	REGION Główny błąd - wszystkie pętle nie działają
	  //kasowanie wartości zmiennych errorStatus odblokowanie magistrali
	  IF "setErrorModbsmasterABB_1" AND "setErrorModbsmasterFal" THEN
	    //ustaw znacznik błędu
	    "db10datablock".setRTU_Error := TRUE;
	    // resetuj mdbusMastererror dla wszystkich pętli
	    "dbTags_master_Fal_1".modbusMaster.error := FALSE;
	    "dbTags_master_ABB_1".modbusMaster.error := FALSE;
	    
	  ELSE
	    "db10datablock".setRTU_Error := FALSE;
	    ;
	  END_IF;
	  
	END_REGION
	
	IF ("db10datablock".RTU_Fal_1errorStatus = 0) AND ("db10datablock".RTU_MPP04_1errorStatus = 0) THEN
	  // kasowanie znacznika błędu komunikacj modbus rtu
	  "db10datablock".setRTU_Error := FALSE;
	  ;
	END_IF;
	
	
	
	
	
	REGION Falownik Modbau RTU
	  // Sprawdzanie czy 
	  IF "dbTags_master_Fal_1".step = 27 THEN
	    // Statement section IF
	    "dbTags_master_Fal_1".modbusMaster.error := FALSE;
	    "dbTags_master_Fal_1".modbusMaster.busy := FALSE;
	    "dbTags_master_Fal_1".modbusMaster.status:= 0;
	    
	   
	   // jeśli MPP04_1 kod błedu 80C8 (brak urządzenia na linni) to uruchom pętlę modbus dla falownika
	    IF "dbTags_master_ABB_1".modbusMaster.status = 16#80C8 AND ("dbTags_master_Fal_1".step = 27 OR "dbTags_master_Fal_1".step = 25 )
	    THEN
	      // Statement section 
	      "setErrorModbsmasterFal" := FALSE;
	      "dbTags_master_Fal_1".step := 1;
	      
	      ;
	    END_IF;
	    
	    ;
	  END_IF;
	  
	  // awaria komunikacji z falownikiem Modbus-RTU
	  IF "setErrorModbsmasterFal" THEN
	    // ustaw bit awarii 
	    "dbmanagement".sterowanie_1.awaria_modbus_falownik:= TRUE
	    ;
	  END_IF;
	  
	  // kasowanie biti awarii komunikacji falownika Modbus-RTU
	  IF "memStep_errorFal" = 100 THEN
	    // kasowanie
	    "dbmanagement".sterowanie_1.awaria_modbus_falownik:= FALSE
	    ;
	  END_IF;
	  
	  
	END_REGION
	
	REGION MPP04-1 Modbau RTU
	  // Sprawdzanie czy 
	  IF "dbTags_master_ABB_1".step = 27 AND "dbTags_master_Fal_1".step = 27
	     THEN
	    // 
	    "dbTags_master_ABB_1".modbusMaster.error := FALSE;
	    "dbTags_master_ABB_1".modbusMaster.busy := FALSE;
	    "dbTags_master_ABB_1".modbusMaster.status := 0;
	    "dbTags_master_Fal_1".step := 1;
	    
	    ;
	  END_IF;
	  
	  IF "dbTags_master_ABB_1".step = 27
	  THEN
	    // 
	    "dbTags_master_ABB_1".modbusMaster.error := FALSE;
	    "dbTags_master_ABB_1".modbusMaster.busy := FALSE;
	    "dbTags_master_ABB_1".modbusMaster.status := 0;
	    //"dbTags_master_MPP04_1".step := 25;
	    
	    ;
	  END_IF;
	  
	  
	  // awaria komunikacji z MPO04 Modbus-RTU
	  IF "setErrorModbsmasterABB_1"  THEN
	    // ustaw bit awarii po czasie zwłoki 
	    "IEC_Timer_errorRTU_histereza_DB".TON(IN:="setErrorModbsmasterABB_1",
	                                          PT:=T#30S);
	    #set_error_RTU := "IEC_Timer_errorRTU_histereza_DB".Q;
	    "dbmanagement".sterowanie_1.awaria_modbus_przepływ_pomp := #set_error_RTU;
	  ELSE
	    #set_error_RTU := FALSE;
	    ;
	  END_IF;
	  
	  // kasowanie biti awarii komunikacjiModbus-RTU
	  IF "memStep_errorMPP04-1" = 100  AND "setErrorModbsmasterABB_1" = FALSE THEN
	    // kasowanie
	    "dbmanagement".sterowanie_1.awaria_modbus_przepływ_pomp:= FALSE
	    ;
	  END_IF;
	  
	END_REGION
	
	
	
	//Modbus RTU Error Code RESET
	REGION Modbus RTU Error Code
	  // Ustaw reset modbus rtu
	  IF "db10datablock".RTU_stepRESET THEN
	    // Ustawienie domyślnych satrtowych 
	    "dbTags_master_ABB_1".step := 1;
	    
	    "dbTags_master_Fal_1".step := 25;
	    "dbTags_slave_RTU".step := 25;
	    
	    // Zerowanie kodu błędu
	    "dbTags_master_ABB_1".modbusMaster.errorStatus := 0;
	    "dbTags_master_Fal_1".modbusMaster.errorStatus := 0;
	    "dbTags_slave_RTU".modbusMaster.errorStatus := 0;
	    
	    "db10datablock".RTU_stepRESET := 0;
	    ;
	  END_IF;
	  
	  
	END_REGION
	
	// Ustawienie Błędu Modbus RTU 
	REGION Set Fault Modbus RTU 
	  // Jeśli zmienna kodu błędu różna od 0 to ustaw znacznik błędu Modbus w bloku danych SCADA
	  // i przekaż wartość błędów
	  IF "dbmanagement".sterowanie_1."alarm-modbus" = TRUE
	    
	  THEN
	    
	    "db10datablock".RTU_MPP04_1errorStatus := "dbTags_master_ABB_1".modbusMaster.errorStatus;
	    // Trzeba dopisać przekazanie błędu z PLC Zasuwy
	   // "DB10_instance_SCADA".RTU_MPP04_2errorStatus := "dbTags_master_MPP04_2".modbusMaster.errorStatus;
	    "db10datablock".RTU_Fal_1errorStatus := "dbTags_master_Fal_1".modbusMaster.errorStatus;
	    "db10datablock".RTU_MT101 := "dbTags_slave_RTU".modbusMaster.errorStatus;
	  ELSE
	    //
	    ;
	    ;
	  END_IF;
	  
	  
	  // Modbus przekaż bit do instancji SCADA Alarm ostrzeżenie kłoport z Modbau
	  // Przynajmniej jeden slave nie odpowiada
	  IF "dbTags_master_Fal_1".step = 27 OR "dbTags_master_ABB_1".step = 27 
	 
	  THEN
	    "dbmanagement".sterowanie_1."alarm-warning" := TRUE;
	
	    ;
	    
	  END_IF;
	  
	  IF "db10datablock".RTU_Fal_1errorStatus = 0 AND "db10datablock".RTU_MPP04_1errorStatus = 0 THEN
	  // kasuj ostrzeżenie
	    "dbmanagement".sterowanie_1."alarm-warning" := FALSE;
	    ;
	  ;
	END_IF;
	
	  
	  
	  
	  
	END_REGION
	
	
	
	
	
END_FUNCTION

FUNCTION_BLOCK "06_M_control strategy Z11"
TITLE = Strategia sterowania 
{ S7_Optimized_Access := 'TRUE' }
AUTHOR : rtecmer
VERSION : 0.1
//Funkcja sterowania przełączaniem kieunku pompowania Z11 - przetłaczania kierunek miasto, Z12 - dosilanie w kierunku magistrali
   VAR_INPUT 
      bit_alarm_magistrala_min { ExternalAccessible := 'False'; ExternalVisible := 'False'; ExternalWritable := 'False'} : Bool := false;   // bit alarmmagistrala awaria niskie ciśnienie
   END_VAR

   VAR_IN_OUT 
      CMD_Open_Z11 : Bool;   // znacznik sterowania otwieraniem
      CMD_Close_Z11 : Bool;   // znacznik sterowania otwieraniem
   END_VAR

   VAR 
      bit_set_open_Z11 { ExternalAccessible := 'False'; ExternalVisible := 'False'; ExternalWritable := 'False'} : Bool;   // bit inicjacji otwierania zasuwy w trybie strategii
      bit_set_open_Z12 { ExternalAccessible := 'False'; ExternalVisible := 'False'; ExternalWritable := 'False'} : Bool;   // bit inicjacji otwierania zasuwy w trybie strategii
      bit_hist_open_Z11 { ExternalAccessible := 'False'; ExternalVisible := 'False'; ExternalWritable := 'False'} : Bool;   // bit opóźnienia reakcji
      bit_hist_open_Z12 { ExternalAccessible := 'False'; ExternalVisible := 'False'; ExternalWritable := 'False'} : Bool;   // bit opóźnienia reakcji
      bit_set_close_Z11 { ExternalAccessible := 'False'; ExternalVisible := 'False'; ExternalWritable := 'False'} : Bool;   // bit inicjacji otwierania zasuwy w trybie strategii
      bit_set_close_Z12 { ExternalAccessible := 'False'; ExternalVisible := 'False'; ExternalWritable := 'False'} : Bool;   // bit inicjacji otwierania zasuwy w trybie strategii
      bit_hist_close_Z11 { ExternalAccessible := 'False'; ExternalVisible := 'False'; ExternalWritable := 'False'} : Bool;   // bit opóźnienia reakcji
      bit_hist_close_Z12 { ExternalAccessible := 'False'; ExternalVisible := 'False'; ExternalWritable := 'False'} : Bool;   // bit opóźnienia reakcji
   END_VAR


BEGIN
	REGION _name_
	  // Statement section REGION
	  
	END_REGION
	(*
	//=============================================================================
	//(JZWiK S.A Radosław Tecmer)
	//(c)Copyright (2021) All Rights Reserved
	//-----------------------------------------------------------------------------
	//Testowane z:   (system docelowy z  FW 4.4)
	//Pakiet inżynierski:   TIA Portal (V14 Sp1 Update 9)
	//Ograniczenia:  ( - )
	//Wymagania:  (minimalne S7-1200 CPU 1215C FW 4.2 .)
	//Funkcjonalnośc: (Sterowanie zasuwą Z11 - miasto, 
	                    Z12 - magistrala. W oparciu o sygnał 
	                   wyboru [dbHoldRegSlave_to_MT101.instSygSter_1 - %DB100.DBW52]
	                   0- wyłączone, 1- dosilanie, 2 - przetłaczanie, 3- automat, 
	                   4- ręczne następuje otwarcie właściwej zasuwy.)
	//-----------------------------------------------------------------------------
	//Zmainy wprowadzone:
	//Wersja  Data       Osoba wprowadzająca zmiany - ekspert
	//01.00.00 17.11.2021 (Tecmer Radosław - twórca) Pieresza wersja 01.00.00
	//=============================================================================
	*)
	
	
	
	
	
	
	
	// Z11 Napełnianie zbiorników
	
	REGION Napełnianie
	  // OTWIERANIE
	  // Warunek wystawienia rozkazu na otwarcie Z1
	  // 
	  IF "Data_Czas_synch".actTime = "dbmanagement".instHourStart_Filling
	    AND "dbtags_Sterowanie"."Paramaetry _Zbiorniki".set_sterowanie_cyklem = 1
	    AND "bitH_REM_Z11"
	    AND "bitH_Aut_Man_Z11"
	    AND "inputOtwartaZ11" = FALSE
	    AND #bit_alarm_magistrala_min = FALSE
	  THEN
	  // 
	    #bit_hist_close_Z11 := FALSE;
	    #CMD_Close_Z11 := FALSE;
	    #bit_hist_open_Z11 := TRUE;
	  ELSE
	    
	  ;
	END_IF;
	
	
	"IEC_Timer_Z11_open_DB".TON(IN:=#bit_hist_open_Z11,
	                            PT:=T#10S,
	                            Q=>#bit_set_open_Z11);
	
	
	IF #bit_set_open_Z11 THEN
	  // start otwieranie
	  #CMD_Open_Z11 := TRUE;
	ELSE
	  #CMD_Open_Z11 := FALSE;
	  ;
	END_IF;
	
	// ZAMYKANIE
	// Warune na zamykanie Z11 gdy zasuwa Z9 zamknięta lub strategia na 1 czyli dosilanie
	// lub pompownia wyłączona 0 
	IF ("maxWaterTank_1" = TRUE OR "maxWaterTank_2" = TRUE  )// poziom max
	  OR #bit_alarm_magistrala_min OR // awaria niskie ciśnienie na magistrali
	  ( "Data_Czas_synch".actTime = "dbmanagement".instHourStop_Filling)
	  AND "bitH_REM_Z11"
	  AND "bitH_Aut_Man_Z11"
	THEN
	  // start zamykanie
	  #bit_hist_open_Z11 := FALSE;
	  #CMD_Open_Z11 := FALSE;
	  #bit_hist_close_Z11:= TRUE;
	ELSE
	  
	  ;
	END_IF;
	
	
	"IEC_Timer_Z11close_DB".TON(IN := #bit_hist_close_Z11,
	                            PT := T#5S,
	                            Q => #bit_set_close_Z11);
	
	
	IF #bit_hist_close_Z11 THEN
	  // start na zamykanie
	  #CMD_Open_Z11 := FALSE;
	  #CMD_Close_Z11 := TRUE;
	ELSE
	  #CMD_Close_Z11 := FALSE;
	  ;
	END_IF;
	
	
	
	END_REGION
	
	REGION Zabezpieczenie przed otwarciem poza czasem napełniania 
	  // nie dopuszczamy do otwarcia zasuwy poza czasem wyznaczonym zakresami strat/stop napełnianie
	  IF ( "Data_Czas_synch".actTime = "dbmanagement".instHourStop_Filling) THEN
	    #bit_hist_open_Z11 := FALSE;
	    #bit_set_open_Z11 := FALSE;
	    #CMD_Open_Z11 := FALSE;
	  
	  ;
	END_IF;
	
	  
	END_REGION
	
	REGION Zabezpieczenie pzy pracy manualnej
	  // blokowanie automatu
	  IF "bitH_Aut_Man_Z11" =  FALSE THEN
	    #bit_hist_open_Z11 := FALSE;
	    ;
	  END_IF;
	  
	  
	END_REGION
	
	
	
	
	
	
	
	
	
END_FUNCTION_BLOCK

FUNCTION_BLOCK "06_M_Alarm-Pomps_value_press"
TITLE = reakcja na niskie ciśnienie na ssaniu
{ S7_Optimized_Access := 'TRUE' }
AUTHOR : rtecmer
VERSION : 0.1
//Funkcja realizuje zatrzymanie pomp z powodu niskiego ciśnienia ssania
   VAR_OUTPUT 
      bit_on_alarm_bar_max_pompownia { ExternalWritable := 'False'} : Bool;   // bit alarmu maksymalnego ciśnienia na pompowni
   END_VAR

   VAR 
      bit_max_pompownia { ExternalAccessible := 'False'; ExternalVisible := 'False'; ExternalWritable := 'False'} : Bool := false;   // bit detekcji wysokiego ciśnienia pompownia B7
      bit_normalne_pompownia { ExternalAccessible := 'False'; ExternalVisible := 'False'; ExternalWritable := 'False'} : Bool := false;   // bit detekcji normalnego cisnienia pompownia
      "bit_max _bar_B7" { ExternalAccessible := 'False'; ExternalVisible := 'False'; ExternalWritable := 'False'} : Bool := false;   // bit zaistnienia max ciśnienia pompownia B7
      bit_off_alarm_max_pompownia { ExternalAccessible := 'False'; ExternalVisible := 'False'; ExternalWritable := 'False'} : Bool;   // koniec alarmu max B7 pompownia
   END_VAR


BEGIN
	(*
	//=============================================================================
	//(JZWiK S.A Radosław Tecmer)
	//(c)Copyright (2021) All Rights Reserved
	//-----------------------------------------------------------------------------
	//Testowane z:   (system docelowy z  FW 4.4)
	//Pakiet inżynierski:   TIA Portal (V14 Sp1 Update 9)
	//Ograniczenia:  ( - )
	//Wymagania:  (minimalne S7-1200 CPU 1215C FW 4.2 .)
	//Funkcjonalnośc: (Kontrola ciśnienia max przepompownia 
	                   Ustawienie i kasowanie bitu awarii od max ciśnienia
	                   na pompowni.)
	//-----------------------------------------------------------------------------
	//Zmainy wprowadzone:
	//Wersja  Data       Osoba wprowadzająca zmiany - ekspert
	//01.00.00 17.11.2021 (Tecmer Radosław - twórca) Pieresza wersja 01.00.00
	//=============================================================================
	*)
	
	
	
	
	
	
	
	
	REGION Kontrola ciśnienia pompownia - ciśnienie max
	  // Kontrola max pompownia ustawione alarmowe 9.0
	  IF "dbdane".act_Value_B5 >= "db10datablock".set_press_bar_Max THEN
	    // Ustaw bit alarmowe ciśnienie na B7
	    #"bit_max _bar_B7" := TRUE;
	    #bit_normalne_pompownia := FALSE;
	  ELSE
	    #bit_normalne_pompownia := TRUE;
	    ;
	  END_IF;
	  
	  
	  //warunek koniec alarmu max
	  IF "dbdane".act_Value_B5 <= ("db10datablock".set_press_bar_Max - 0.2) THEN
	    // ustaw bit ciśnienie poprawne
	    #bit_normalne_pompownia := TRUE;
	    ;
	  END_IF;
	  
	  // kasowania alarmu
	  IF #bit_off_alarm_max_pompownia THEN
	    // kasowanie alarmu ssania
	    #bit_on_alarm_bar_max_pompownia := FALSE;
	    #"bit_max _bar_B7" := FALSE;
	    
	  END_IF;
	  
	  // Histerez ana ustawienie alarmu max bar
	  "IEC_Timer_B7max_bar_DB".TON(IN:=#"bit_max _bar_B7",
	                               PT:=T#10S,
	                               Q=>#bit_on_alarm_bar_max_pompownia);
	  
	 "IEC_Timer_B7max_off_alarm_DB".TON(IN:=#bit_normalne_pompownia,
	                                   PT:=T#10S,
	                                   Q=>#bit_off_alarm_max_pompownia);
	
	
	  
	  
	  
	  
	END_REGION
	
	
END_FUNCTION_BLOCK

FUNCTION_BLOCK "06_M_Control strategy Pumping station"   // FB4, LAD
TITLE = Ustawienie metody sterowania
{ S7_Optimized_Access := 'TRUE' }
AUTHOR : rtecmer
VERSION : 0.1
// stored: AutoNumber true, IsIECCheckEnabled false, IsRetainMemResEnabled false, MemoryReserve 100, SetENOAutomatically false, UDAEnableTagReadback false
   VAR_INPUT
      tempStrategia_Pompownia : Int;   // Słowo strategii przechwyconej w FB24
      "bit_alarm_magistrala _min" : Bool;   // bit alarmu niskie ciśniei na magistrali
      bit_off_alarm_magistrala_niskie : Bool;   // bit wyłaczenia alarmu magistrali niskie
   END_VAR
   VAR_IN_OUT
      "Strategia Pompownia" : Int;
   END_VAR
   VAR
      tmp_on_alarm { ExternalAccessible := 'False'; ExternalVisible := 'False'; ExternalWritable := 'False'} : Bool;
      tmp_off_alarm { ExternalAccessible := 'False'; ExternalVisible := 'False'; ExternalWritable := 'False'} : Bool;
      memTriger_set_Strategia { ExternalAccessible := 'False'; ExternalVisible := 'False'; ExternalWritable := 'False'} : Bool;
      memTriger_reset_Strategia { ExternalAccessible := 'False'; ExternalVisible := 'False'; ExternalWritable := 'False'} : Bool;
      test { ExternalAccessible := 'False'; ExternalVisible := 'False'; ExternalWritable := 'False'} : Bool;
   END_VAR
   VAR CONSTANT
      "strategia awaria" : Int := 0;   // regulator wyłączony gdy brak wody w zbiornikach i małae ciśnienie na magistrali
   END_VAR
   VAR_TEMP   // added for the SCL form of the ladder/FBD networks
      _w1 : Bool;
      _w2 : Bool;
   END_VAR
BEGIN

REGION Network 1: Koniec awarii magistrali
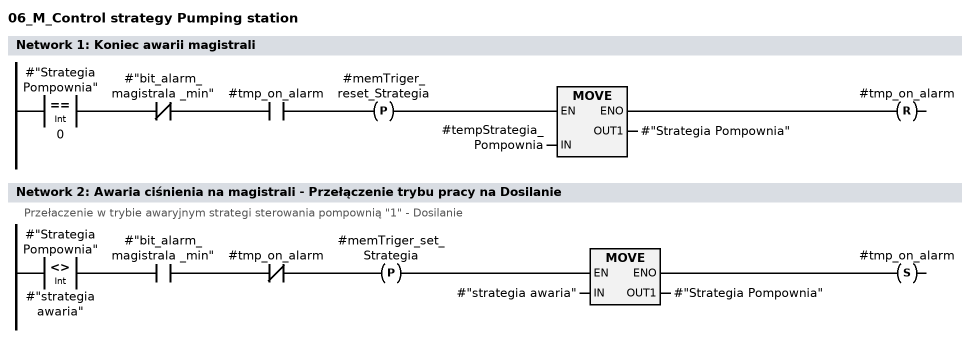
   RUNG wire#powerrail
      { S7_Templates := "SrcType := Int" } EQ_Contact(in1 := #"Strategia Pompownia", in2 := 0)
      I_Contact( #"bit_alarm_magistrala _min" )
      Contact( #tmp_on_alarm )
      P_Trig( #memTriger_reset_Strategia )
      Move(in := #tempStrategia_Pompownia, out1 => #"Strategia Pompownia")
      R_Coil( #tmp_on_alarm )
   END_RUNG
   // the same network as SCL:
   #_w1 := (#"Strategia Pompownia" = 0) AND NOT #"bit_alarm_magistrala _min" AND #tmp_on_alarm;
   #_w2 := #_w1 AND NOT #memTriger_reset_Strategia;   // rising edge
   #memTriger_reset_Strategia := #_w1;
   IF #_w2 THEN
       #"Strategia Pompownia" := #tempStrategia_Pompownia;
       #tmp_on_alarm := FALSE;
   END_IF;
END_REGION

REGION Network 2: Awaria ciśnienia na magistrali - Przełączenie trybu pracy na Dosilanie
   // Przełaczenie w trybie awaryjnym strategi sterowania pompownią "1" - Dosilanie
   RUNG wire#powerrail
      { S7_Templates := "SrcType := Int" } NE_Contact(in1 := #"Strategia Pompownia", in2 := #"strategia awaria")
      Contact( #"bit_alarm_magistrala _min" )
      I_Contact( #tmp_on_alarm )
      P_Trig( #memTriger_set_Strategia )
      Move(in := #"strategia awaria", out1 => #"Strategia Pompownia")
      S_Coil( #tmp_on_alarm )
   END_RUNG
   // the same network as SCL:
   #_w1 := (#"Strategia Pompownia" <> #"strategia awaria") AND #"bit_alarm_magistrala _min" AND NOT #tmp_on_alarm;
   #_w2 := #_w1 AND NOT #memTriger_set_Strategia;   // rising edge
   #memTriger_set_Strategia := #_w1;
   IF #_w2 THEN
       #"Strategia Pompownia" := #"strategia awaria";
       #tmp_on_alarm := TRUE;
   END_IF;
END_REGION
END_FUNCTION_BLOCK

FUNCTION_BLOCK "00_S_VLV02"   // FB5, LAD
TITLE = Valve driver 02
{ S7_Optimized_Access := 'FALSE' }
AUTHOR : RTecmer
VERSION : 0.2
// Driver for two-position drives
// Slowo STATUSU Napedu
// STAT - Prawy Byte
// WIZ  - Lewy Byte
//  
//   -STAT wektor stanu zaworu
//     -bit 0- alarm                                  (sygnal do SCADA)
//     -bit 1- zawor otwarty                    (sygnal do SCADA)
//     -bit 2-sterowanie zdal=1 loc=0 (sygnal do SCADA)
//     -bit 3- zawor zamkniety               (sygnal do SCADA)
//     -bit 4-otwieranie reczne              (sygnal z SCADA)
//     -bit 5-zamykanie reczne              (sygnal z SCADA)
//     -bit 6-alarm reset                        (sygnal z SCADA
//     -bit 8-auto= 1man=0                  (sygnal z SCADA)
//   -SUPV 
//   -CLSD zawor zamkniety                    - wejscie
//   -OPND zawor otwarty                        - wejscie
//   -REMT sterowanie zdal=1 loc=0      - wejscie
//   -OPEN otwarcie                                  - wyjscie
//   -CLSE zamkniecie                              - wyjscie
//   - TIM1 czas otwierania  
//   - TIM2 czas zamykania
// stored: AutoNumber true, IsIECCheckEnabled false, SetENOAutomatically false, UDAEnableTagReadback false
   VAR_INPUT
      SVMC : Bool;   // Automat na zamykanie
      SVMO { ExternalVisible := 'False'} : Bool;   // Automat na otwieranie
      CLSD : Bool;   // Zamknięta
      OPND : Bool;   // Otwarta
      REMT : Bool;   // Sterowanie zdalne =1, remontowe=0
      KT1 : Time;   // Czas timera
   END_VAR
   VAR_IN_OUT
      CLSE { ExternalAccessible := 'False'; ExternalVisible := 'False'; ExternalWritable := 'False'} : Bool;   // Wyjście zamykanie
      OPEN { ExternalAccessible := 'False'; ExternalVisible := 'False'; ExternalWritable := 'False'} : Bool;   // Wyjście Otwieranie
      WIZ : Byte;   // Wektor SCADA
      STAT : Byte;   // Wektor statusu napędu
      TMR1 : TON_TIME;
   END_VAR
BEGIN

REGION Network 1
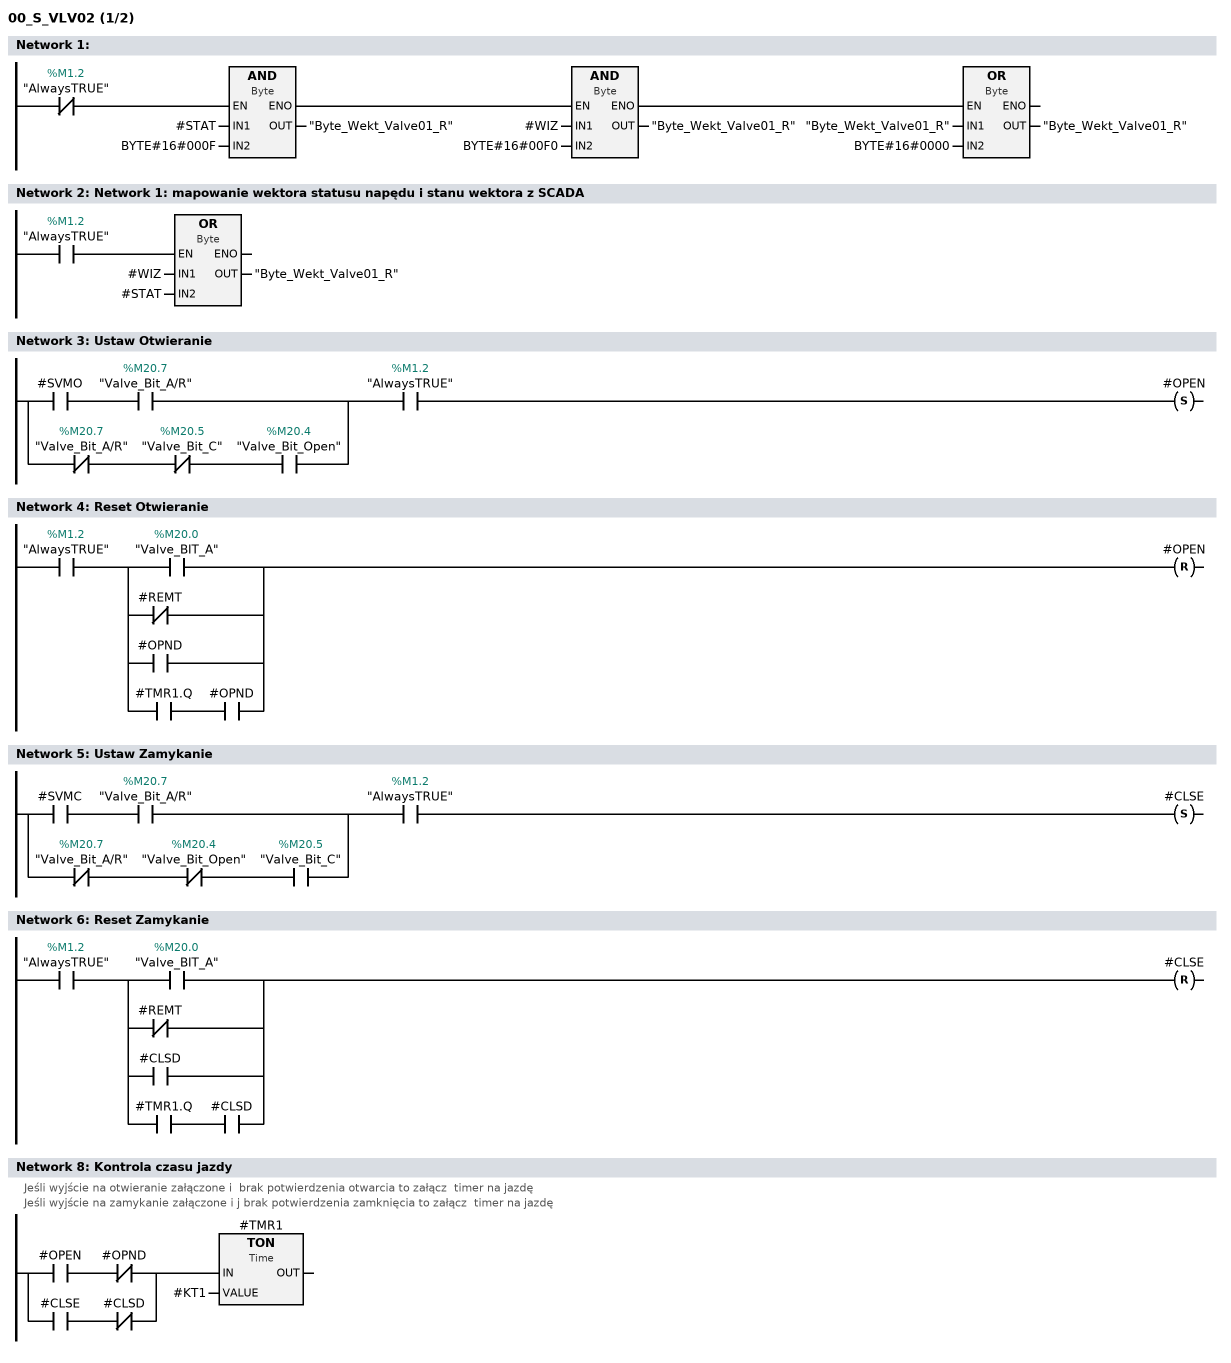
   IF NOT "AlwaysTRUE" THEN
       "Byte_Wekt_Valve01_R" := #STAT AND BYTE#16#000F;
       "Byte_Wekt_Valve01_R" := #WIZ AND BYTE#16#00F0;
       "Byte_Wekt_Valve01_R" := "Byte_Wekt_Valve01_R" OR BYTE#16#0000;
   END_IF;
END_REGION

REGION Network 2: Network 1: mapowanie wektora statusu napędu i stanu wektora z SCADA
   IF "AlwaysTRUE" THEN "Byte_Wekt_Valve01_R" := #WIZ OR #STAT; END_IF;
END_REGION

REGION Network 3: Ustaw Otwieranie
   RUNG wire#powerrail
      Contact( #SVMO )
      Contact( "Valve_Bit_A/R" )
      wire#w1
      Contact( "AlwaysTRUE" )
      S_Coil( #OPEN )
   END_RUNG
   RUNG wire#powerrail
      I_Contact( "Valve_Bit_A/R" )
      I_Contact( "Valve_Bit_C" )
      Contact( "Valve_Bit_Open" )
   END_RUNG wire#w1
   // the same network as SCL:
   IF ((#SVMO AND "Valve_Bit_A/R") OR (NOT "Valve_Bit_A/R" AND NOT "Valve_Bit_C" AND "Valve_Bit_Open")) AND "AlwaysTRUE" THEN
       #OPEN := TRUE;
   END_IF;
END_REGION

REGION Network 4: Reset Otwieranie
   RUNG wire#powerrail
      Contact( "AlwaysTRUE" )
      wire#w1
      Contact( "Valve_BIT_A" )
      wire#w2
      R_Coil( #OPEN )
   END_RUNG
   RUNG wire#w1
      I_Contact( #REMT )
   END_RUNG wire#w2
   RUNG wire#w1
      Contact( #OPND )
   END_RUNG wire#w2
   RUNG wire#w1
      Contact( #TMR1.Q )
      Contact( #OPND )
   END_RUNG wire#w2
   // the same network as SCL:
   IF "AlwaysTRUE" AND ("Valve_BIT_A" OR NOT #REMT OR #OPND OR (#TMR1.Q AND #OPND)) THEN
       #OPEN := FALSE;
   END_IF;
END_REGION

REGION Network 5: Ustaw Zamykanie
   RUNG wire#powerrail
      Contact( #SVMC )
      Contact( "Valve_Bit_A/R" )
      wire#w1
      Contact( "AlwaysTRUE" )
      S_Coil( #CLSE )
   END_RUNG
   RUNG wire#powerrail
      I_Contact( "Valve_Bit_A/R" )
      I_Contact( "Valve_Bit_Open" )
      Contact( "Valve_Bit_C" )
   END_RUNG wire#w1
   // the same network as SCL:
   IF ((#SVMC AND "Valve_Bit_A/R") OR (NOT "Valve_Bit_A/R" AND NOT "Valve_Bit_Open" AND "Valve_Bit_C")) AND "AlwaysTRUE" THEN
       #CLSE := TRUE;
   END_IF;
END_REGION

REGION Network 6: Reset Zamykanie
   RUNG wire#powerrail
      Contact( "AlwaysTRUE" )
      wire#w1
      Contact( "Valve_BIT_A" )
      wire#w2
      R_Coil( #CLSE )
   END_RUNG
   RUNG wire#w1
      I_Contact( #REMT )
   END_RUNG wire#w2
   RUNG wire#w1
      Contact( #CLSD )
   END_RUNG wire#w2
   RUNG wire#w1
      Contact( #TMR1.Q )
      Contact( #CLSD )
   END_RUNG wire#w2
   // the same network as SCL:
   IF "AlwaysTRUE" AND ("Valve_BIT_A" OR NOT #REMT OR #CLSD OR (#TMR1.Q AND #CLSD)) THEN
       #CLSE := FALSE;
   END_IF;
END_REGION

REGION Network 8: Kontrola czasu jazdy
   // Jeśli wyjście na otwieranie załączone i  brak potwierdzenia otwarcia to załącz  timer na jazdę
   // Jeśli wyjście na zamykanie załączone i j brak potwierdzenia zamknięcia to załącz  timer na jazdę
   #TMR1(IN := (#OPEN AND NOT #OPND) OR (#CLSE AND NOT #CLSD), PT := #KT1);   // TON coil
END_REGION

REGION Network 9: Bit alarm ustaw
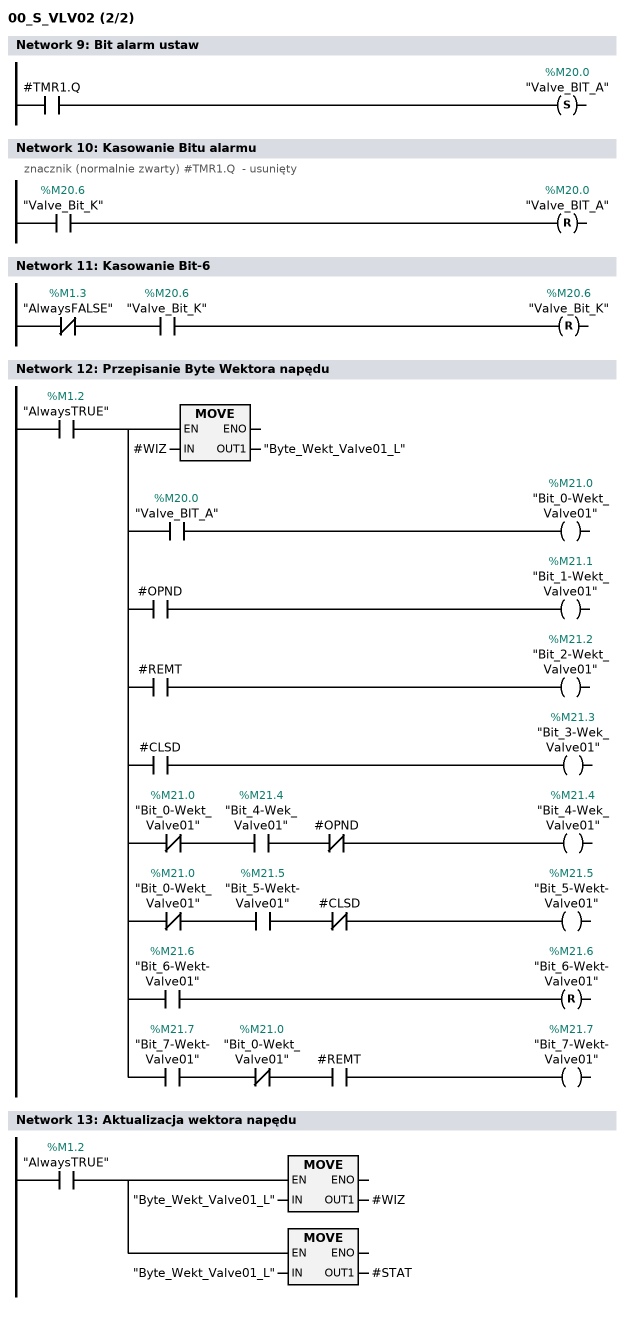
   RUNG wire#powerrail
      Contact( #TMR1.Q )
      S_Coil( "Valve_BIT_A" )
   END_RUNG
   // the same network as SCL:
   IF #TMR1.Q THEN "Valve_BIT_A" := TRUE; END_IF;
END_REGION

REGION Network 10: Kasowanie Bitu alarmu
   // znacznik (normalnie zwarty) #TMR1.Q  - usunięty
   RUNG wire#powerrail
      Contact( "Valve_Bit_K" )
      R_Coil( "Valve_BIT_A" )
   END_RUNG
   // the same network as SCL:
   IF "Valve_Bit_K" THEN "Valve_BIT_A" := FALSE; END_IF;
END_REGION

REGION Network 11: Kasowanie Bit-6
   RUNG wire#powerrail
      I_Contact( "AlwaysFALSE" )
      Contact( "Valve_Bit_K" )
      R_Coil( "Valve_Bit_K" )
   END_RUNG
   // the same network as SCL:
   IF NOT "AlwaysFALSE" AND "Valve_Bit_K" THEN "Valve_Bit_K" := FALSE; END_IF;
END_REGION

REGION Network 12: Przepisanie Byte Wektora napędu
   RUNG wire#powerrail
      Contact( "AlwaysTRUE" )
      wire#w1
      { S7_GenerateENO := "TRUE" } Move(in := #WIZ, out1 => "Byte_Wekt_Valve01_L")
   END_RUNG
   RUNG wire#w1
      Contact( "Valve_BIT_A" )
      Coil( "Bit_0-Wekt_Valve01" )
   END_RUNG
   RUNG wire#w1
      Contact( #OPND )
      Coil( "Bit_1-Wekt_Valve01" )
   END_RUNG
   RUNG wire#w1
      Contact( #REMT )
      Coil( "Bit_2-Wekt_Valve01" )
   END_RUNG
   RUNG wire#w1
      Contact( #CLSD )
      Coil( "Bit_3-Wek_Valve01" )
   END_RUNG
   RUNG wire#w1
      I_Contact( "Bit_0-Wekt_Valve01" )
      Contact( "Bit_4-Wek_Valve01" )
      I_Contact( #OPND )
      Coil( "Bit_4-Wek_Valve01" )
   END_RUNG
   RUNG wire#w1
      I_Contact( "Bit_0-Wekt_Valve01" )
      Contact( "Bit_5-Wekt-Valve01" )
      I_Contact( #CLSD )
      Coil( "Bit_5-Wekt-Valve01" )
   END_RUNG
   RUNG wire#w1
      Contact( "Bit_6-Wekt-Valve01" )
      R_Coil( "Bit_6-Wekt-Valve01" )
   END_RUNG
   RUNG wire#w1
      Contact( "Bit_7-Wekt-Valve01" )
      I_Contact( "Bit_0-Wekt_Valve01" )
      Contact( #REMT )
      Coil( "Bit_7-Wekt-Valve01" )
   END_RUNG
   // the same network as SCL:
   IF "AlwaysTRUE" THEN "Byte_Wekt_Valve01_L" := #WIZ; END_IF;
   "Bit_0-Wekt_Valve01" := "AlwaysTRUE" AND "Valve_BIT_A";
   "Bit_1-Wekt_Valve01" := "AlwaysTRUE" AND #OPND;
   "Bit_2-Wekt_Valve01" := "AlwaysTRUE" AND #REMT;
   "Bit_3-Wek_Valve01" := "AlwaysTRUE" AND #CLSD;
   "Bit_4-Wek_Valve01" := "AlwaysTRUE" AND NOT "Bit_0-Wekt_Valve01" AND "Bit_4-Wek_Valve01" AND NOT #OPND;
   "Bit_5-Wekt-Valve01" := "AlwaysTRUE" AND NOT "Bit_0-Wekt_Valve01" AND "Bit_5-Wekt-Valve01" AND NOT #CLSD;
   IF "AlwaysTRUE" AND "Bit_6-Wekt-Valve01" THEN "Bit_6-Wekt-Valve01" := FALSE; END_IF;
   "Bit_7-Wekt-Valve01" := "AlwaysTRUE" AND "Bit_7-Wekt-Valve01" AND NOT "Bit_0-Wekt_Valve01" AND #REMT;
END_REGION

REGION Network 13: Aktualizacja wektora napędu
   RUNG wire#powerrail
      Contact( "AlwaysTRUE" )
      wire#w1
      { S7_GenerateENO := "TRUE" } Move(in := "Byte_Wekt_Valve01_L", out1 => #WIZ)
   END_RUNG
   RUNG wire#w1
      { S7_GenerateENO := "TRUE" } Move(in := "Byte_Wekt_Valve01_L", out1 => #STAT)
   END_RUNG
   // the same network as SCL:
   IF "AlwaysTRUE" THEN
       #WIZ := "Byte_Wekt_Valve01_L";
       #STAT := "Byte_Wekt_Valve01_L";
   END_IF;
END_REGION
END_FUNCTION_BLOCK

FUNCTION_BLOCK "08_M_Converting parameters from the inverter"
{ S7_Optimized_Access := 'TRUE' }
AUTHOR : rtecmer
VERSION : 0.1
   VAR_INPUT 
      received_Inver_setpoint_ref_416020 { ExternalAccessible := 'False'; ExternalVisible := 'False'; ExternalWritable := 'False'} : Int;
      received_Inver_Frequency_416130 { ExternalAccessible := 'False'; ExternalVisible := 'False'; ExternalWritable := 'False'} : Int;
      received_Inver_MotorCurrent_416140 { ExternalAccessible := 'False'; ExternalVisible := 'False'; ExternalWritable := 'False'} : Int;
      received_Inver_NomCurrent_416360 { ExternalAccessible := 'False'; ExternalVisible := 'False'; ExternalWritable := 'False'} : Int;
      received_Inver_MaxCurrent_416370 { ExternalAccessible := 'False'; ExternalVisible := 'False'; ExternalWritable := 'False'} : Int;
      received_Inver_InDigit_416600 { ExternalAccessible := 'False'; ExternalVisible := 'False'; ExternalWritable := 'False'} : Int;
      received_Inver_OverTemp_415040 { ExternalAccessible := 'False'; ExternalVisible := 'False'; ExternalWritable := 'False'} : Int;
      received_Inver_OverVolts_415050 { ExternalAccessible := 'False'; ExternalVisible := 'False'; ExternalWritable := 'False'} : Int;
   END_VAR

   VAR_OUTPUT 
      Setpoint_Inverter { ExternalAccessible := 'False'; ExternalVisible := 'False'; ExternalWritable := 'False'} : Real;   // Wartość zadana Hz odczytane z Modbus
      Frequency_inverter { ExternalAccessible := 'False'; ExternalVisible := 'False'; ExternalWritable := 'False'} : Real;   // Aktualne Hz silniku odczytane z Modbus
      MotorCurrent_Inverter { ExternalAccessible := 'False'; ExternalVisible := 'False'; ExternalWritable := 'False'} : Real;   // Prąd na silniku zasilanym z falownika odczytane z Modbus
      NormalCurrent_Inverter { ExternalAccessible := 'False'; ExternalVisible := 'False'; ExternalWritable := 'False'} : Real;   // Prąd nominalny falownika odczytane z Modbus
      MaxCurrent_Inverter { ExternalAccessible := 'False'; ExternalVisible := 'False'; ExternalWritable := 'False'} : Real;   // Prad Max krótkotrwały odczytane z Modbus
      OverTemp_Inverter { ExternalAccessible := 'False'; ExternalVisible := 'False'; ExternalWritable := 'False'} : Word;
      OverVolta_Inverter { ExternalAccessible := 'False'; ExternalVisible := 'False'; ExternalWritable := 'False'} : Word;
   END_VAR

   VAR 
      tmp_1 { ExternalAccessible := 'False'; ExternalVisible := 'False'; ExternalWritable := 'False'} : Real;
      tmp_2 { ExternalAccessible := 'False'; ExternalVisible := 'False'; ExternalWritable := 'False'} : Real;
      tmp_3 { ExternalAccessible := 'False'; ExternalVisible := 'False'; ExternalWritable := 'False'} : Real;
      tmp_4 { ExternalAccessible := 'False'; ExternalVisible := 'False'; ExternalWritable := 'False'} : Real;
      tmp_5 { ExternalAccessible := 'False'; ExternalVisible := 'False'; ExternalWritable := 'False'} : Real;
      tmp_6 { ExternalAccessible := 'False'; ExternalVisible := 'False'; ExternalWritable := 'False'} : Real;
      tmp_7 { ExternalAccessible := 'False'; ExternalVisible := 'False'; ExternalWritable := 'False'} : Real;
      tmp_8 { ExternalAccessible := 'False'; ExternalVisible := 'False'; ExternalWritable := 'False'} : Real;
      tmp_9 { ExternalAccessible := 'False'; ExternalVisible := 'False'; ExternalWritable := 'False'} : Real;
      tmp_10 { ExternalAccessible := 'False'; ExternalVisible := 'False'; ExternalWritable := 'False'} : Real;
   END_VAR


BEGIN
	(*
	//=============================================================================
	//(JZWiK S.A Radosław Tecmer)
	//(c)Copyright (2021) All Rights Reserved
	//-----------------------------------------------------------------------------
	//Testowane z:   (system docelowy z  FW 4.4)
	//Pakiet inżynierski:   TIA Portal (V14 Sp1 Update 9)
	//Ograniczenia:  ( - )
	//Wymagania:  (minimalne S7-1200 CPU 1215C FW 4.2 .)
	//Funkcjonalnośc: (Konwersja i przeliczenie wartości pobranych  z Modbus RTU 
	//                  na wartości rzeczywiste)
	//-----------------------------------------------------------------------------
	//Zmainy wprowadzone:
	//Wersja  Data       Osoba wprowadzająca zmiany - ekspert
	//01.00.00 11.01.2022 (Tecmer Radosław - twórca) Pieresza wersja 01.00.00
	//=============================================================================
	*)
	
	
	//Wartości indexów zgodnie z dokumentacją Danfoss FC51 Programing Guide:
	//index 2 | mnożnik 10; index 1 | mnożnik 100; index 0 | mnożnik 0
	//index -1 | mnożnik 0.1; index -2 | mnożnik 0.01; index -3 | mnożnik 0.001
	//index -4 | mnożnik 0.0001; index -5 | mnożnik 0.00001
	
	REGION Setpoint Inverter P1-P4
	  // Wyliczanie wartości 
	  #tmp_1 := INT_TO_REAL (#received_Inver_setpoint_ref_416020 );
	  #tmp_2 := (#tmp_1 * 0.1) * 0.01;
	  #Setpoint_Inverter := SCALE_X_REAL(MIN := 0.0,
	                                           VALUE := #tmp_2,
	                                           MAX := 50.0);
	  
	END_REGION
	
	REGION Frequecy Act. Inverter P1-P4
	  // Wyliczanie wartości
	  #tmp_3 := INT_TO_REAL(#received_Inver_Frequency_416130) ;
	  #tmp_4 := (#tmp_3 * 0.1);
	  #Frequency_inverter := #tmp_4;
	  
	END_REGION
	
	REGION Motor Current from Inverter P1-P4
	  // Wyliczanie wartości
	  #tmp_5 := INT_TO_REAL(#received_Inver_MotorCurrent_416140);
	  #tmp_6 := (#tmp_5 * 0.01);
	  #MotorCurrent_Inverter := #tmp_6;
	  
	END_REGION
	
	REGION Nominal Current Inverter P1-P4
	  // Wyliczanie wartości
	  #tmp_7 := INT_TO_REAL(#received_Inver_NomCurrent_416360 );
	  #tmp_8 := (#tmp_7 * 0.01);
	  #NormalCurrent_Inverter := #tmp_8;
	  
	END_REGION
	
	REGION Max Current Inverter P1-P4
	  // Wyliczanie wartości
	  #tmp_9 := INT_TO_REAL(#received_Inver_MaxCurrent_416370 );
	  #tmp_10 := (#tmp_9 * 0.01);
	  #MaxCurrent_Inverter := #tmp_10;
	  
	END_REGION
	
	
	#OverTemp_Inverter:= #received_Inver_OverTemp_415040;
	#OverVolta_Inverter:= #received_Inver_OverVolts_415050;
	
	
END_FUNCTION_BLOCK

FUNCTION_BLOCK "06_M_control without inverter"   // FB18, LAD
TITLE = Sterowania bez falownika
{ S7_Optimized_Access := 'TRUE' }
AUTHOR : rtecmer
VERSION : 0.1
// Sterowanie awaryjne układemw w wypadku awarii falownika.
// Sterowanie napędami z sieci. 
// Załączenie od sygnału  InputWarning_L_PID. jest to bit ustawiany przez regulator PID  wyliczany na podstawie wartości zadanej bar + wartość współczynnika .
// Wyłaczenie natępuje po osiągnięciu "Górnego progu tymczasowego". 
// Praca kompresorów z wyrównaniem liczników pracy.
// Jednocześnie pracuje tylko jeden kompresor.
// stored: AutoNumber true, IsIECCheckEnabled false, IsRetainMemResEnabled false, MemoryReserve 500, SetENOAutomatically false, UDAEnableTagReadback false
   VAR_INPUT
      IsReadyP1 : Bool;   // Gotowość pompy
      IsReadyP2 : Bool;   // Gotowość pompy
      IsReadyP3 : Bool;   // Gotowość pompy
      IsReadyP4 : Bool;
      IsMode_Auto : Bool;   // Tryb pracy Aut
      InputWarning_H_PID : Bool;   // Oszczerzenie górny limit
      InputWarning_L_PID : Bool;   // Oczszczerzenie dolny limit
      IsReady_Inverter : Bool;   // Gotowość falownika
      PV_max : Real;   // Wartość górnego progu ostrzegawczego
      Act_B3ciśnienie : Real;   // Aktualna wartość bar
      Rst_Driver_Max_presure : Bool;   // Znacznika awaryjnego wyłączenia od max ciśnienia napędu pracującego w trybie awaryjnym
   END_VAR
   VAR_OUTPUT
      CMD_A_Network_P1 : Bool;   // Bit startu pompyw trybie awaryjnym na soft-startcie
      CMD_A_Network_P2 : Bool := false;   // Bit startu pompyw trybie awaryjnym na soft-startcie
      CMD_A_Network_P3 : Bool := false;   // Bit startu pompyw trybie awaryjnym na soft-startcie
      CMD_A_Network_P4 : Bool := false;   // Bit startu pompyw trybie awaryjnym na soft-startcie
   END_VAR
   VAR
      stc_PV : Real := 0.2;   // Ustalona wartość pomniejszenia PV
   END_VAR
   VAR_TEMP
      set_Motor : Bool;   // pomocniczy bit ustawiający pompę
      tmp_PVmax : Real;   // Tymczasowa ustalona wartość progu górnego bar
   END_VAR
BEGIN

REGION Network 2: Górny próg tymczasowy
   // Wyliczenie górnego progu tymczasowego na potrzeby sterowania wyłączaniem pomp
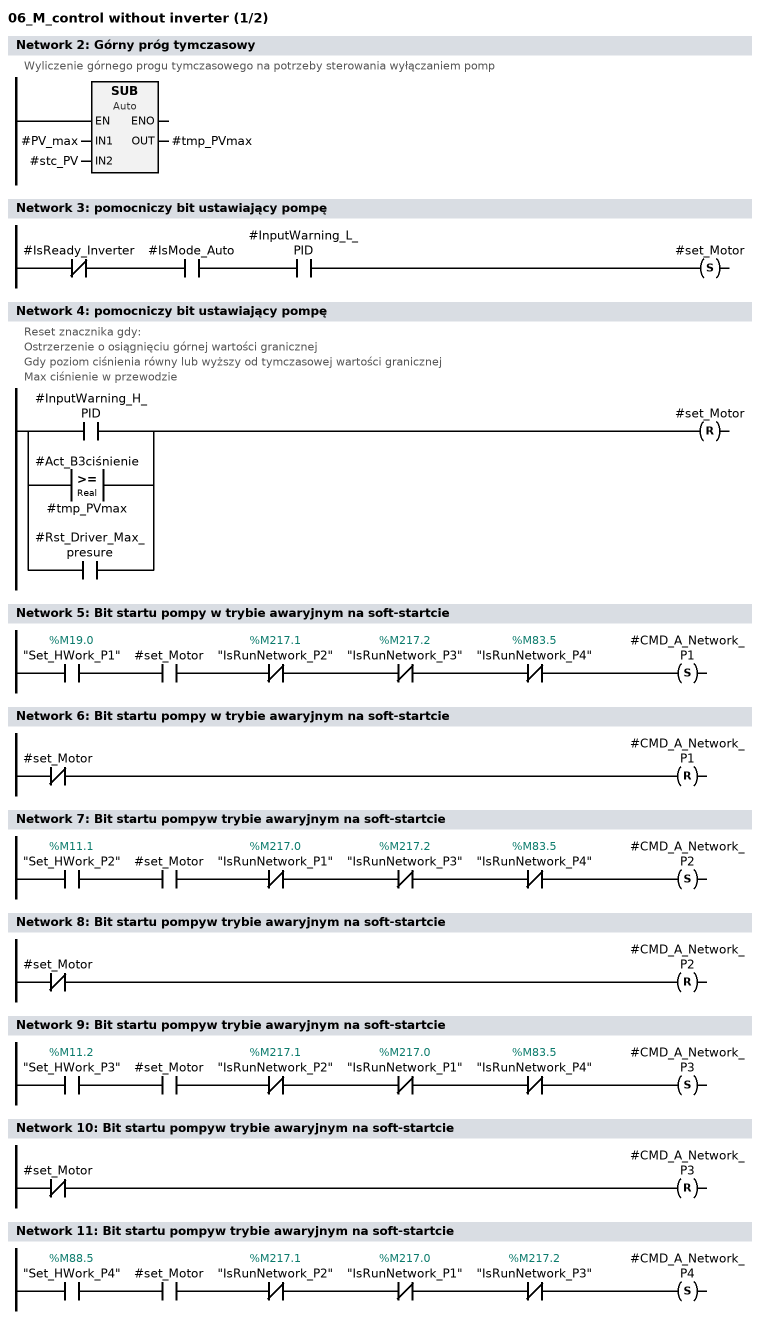
   RUNG wire#powerrail
      Sub(in1 := #PV_max, in2 := #stc_PV, out => #tmp_PVmax)
   END_RUNG
   // the same network as SCL:
   #tmp_PVmax := #PV_max - #stc_PV;
END_REGION

REGION Network 3: pomocniczy bit ustawiający pompę
   RUNG wire#powerrail
      I_Contact( #IsReady_Inverter )
      Contact( #IsMode_Auto )
      Contact( #InputWarning_L_PID )
      S_Coil( #set_Motor )
   END_RUNG
   // the same network as SCL:
   IF NOT #IsReady_Inverter AND #IsMode_Auto AND #InputWarning_L_PID THEN #set_Motor := TRUE; END_IF;
END_REGION

REGION Network 4: pomocniczy bit ustawiający pompę
   // Reset znacznika gdy:
   // Ostrzerzenie o osiągnięciu górnej wartości granicznej
   // Gdy poziom ciśnienia równy lub wyższy od tymczasowej wartości granicznej
   // Max ciśnienie w przewodzie
   RUNG wire#powerrail
      Contact( #InputWarning_H_PID )
      wire#w1
      R_Coil( #set_Motor )
   END_RUNG
   RUNG wire#powerrail
      { S7_Templates := "SrcType := Real" } GE_Contact(in1 := #Act_B3ciśnienie, in2 := #tmp_PVmax)
   END_RUNG wire#w1
   RUNG wire#powerrail
      Contact( #Rst_Driver_Max_presure )
   END_RUNG wire#w1
   // the same network as SCL:
   IF #InputWarning_H_PID OR (#Act_B3ciśnienie >= #tmp_PVmax) OR #Rst_Driver_Max_presure THEN
       #set_Motor := FALSE;
   END_IF;
END_REGION

REGION Network 5: Bit startu pompy w trybie awaryjnym na soft-startcie
   RUNG wire#powerrail
      Contact( "Set_HWork_P1" )
      Contact( #set_Motor )
      I_Contact( "IsRunNetwork_P2" )
      I_Contact( "IsRunNetwork_P3" )
      I_Contact( "IsRunNetwork_P4" )
      S_Coil( #CMD_A_Network_P1 )
   END_RUNG
   // the same network as SCL:
   IF "Set_HWork_P1" AND #set_Motor AND NOT "IsRunNetwork_P2" AND NOT "IsRunNetwork_P3" AND NOT "IsRunNetwork_P4" THEN
       #CMD_A_Network_P1 := TRUE;
   END_IF;
END_REGION

REGION Network 6: Bit startu pompy w trybie awaryjnym na soft-startcie
   RUNG wire#powerrail
      I_Contact( #set_Motor )
      R_Coil( #CMD_A_Network_P1 )
   END_RUNG
   // the same network as SCL:
   IF NOT #set_Motor THEN #CMD_A_Network_P1 := FALSE; END_IF;
END_REGION

REGION Network 7: Bit startu pompyw trybie awaryjnym na soft-startcie
   RUNG wire#powerrail
      Contact( "Set_HWork_P2" )
      Contact( #set_Motor )
      I_Contact( "IsRunNetwork_P1" )
      I_Contact( "IsRunNetwork_P3" )
      I_Contact( "IsRunNetwork_P4" )
      S_Coil( #CMD_A_Network_P2 )
   END_RUNG
   // the same network as SCL:
   IF "Set_HWork_P2" AND #set_Motor AND NOT "IsRunNetwork_P1" AND NOT "IsRunNetwork_P3" AND NOT "IsRunNetwork_P4" THEN
       #CMD_A_Network_P2 := TRUE;
   END_IF;
END_REGION

REGION Network 8: Bit startu pompyw trybie awaryjnym na soft-startcie
   RUNG wire#powerrail
      I_Contact( #set_Motor )
      R_Coil( #CMD_A_Network_P2 )
   END_RUNG
   // the same network as SCL:
   IF NOT #set_Motor THEN #CMD_A_Network_P2 := FALSE; END_IF;
END_REGION

REGION Network 9: Bit startu pompyw trybie awaryjnym na soft-startcie
   RUNG wire#powerrail
      Contact( "Set_HWork_P3" )
      Contact( #set_Motor )
      I_Contact( "IsRunNetwork_P2" )
      I_Contact( "IsRunNetwork_P1" )
      I_Contact( "IsRunNetwork_P4" )
      S_Coil( #CMD_A_Network_P3 )
   END_RUNG
   // the same network as SCL:
   IF "Set_HWork_P3" AND #set_Motor AND NOT "IsRunNetwork_P2" AND NOT "IsRunNetwork_P1" AND NOT "IsRunNetwork_P4" THEN
       #CMD_A_Network_P3 := TRUE;
   END_IF;
END_REGION

REGION Network 10: Bit startu pompyw trybie awaryjnym na soft-startcie
   RUNG wire#powerrail
      I_Contact( #set_Motor )
      R_Coil( #CMD_A_Network_P3 )
   END_RUNG
   // the same network as SCL:
   IF NOT #set_Motor THEN #CMD_A_Network_P3 := FALSE; END_IF;
END_REGION

REGION Network 11: Bit startu pompyw trybie awaryjnym na soft-startcie
   RUNG wire#powerrail
      Contact( "Set_HWork_P4" )
      Contact( #set_Motor )
      I_Contact( "IsRunNetwork_P2" )
      I_Contact( "IsRunNetwork_P1" )
      I_Contact( "IsRunNetwork_P3" )
      S_Coil( #CMD_A_Network_P4 )
   END_RUNG
   // the same network as SCL:
   IF "Set_HWork_P4" AND #set_Motor AND NOT "IsRunNetwork_P2" AND NOT "IsRunNetwork_P1" AND NOT "IsRunNetwork_P3" THEN
       #CMD_A_Network_P4 := TRUE;
   END_IF;
END_REGION

REGION Network 12: Bit startu pompyw trybie awaryjnym na soft-startcie
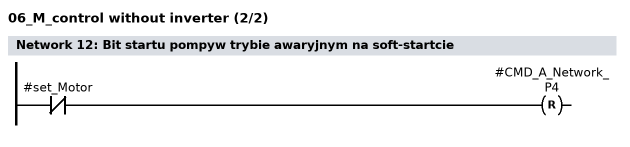
   RUNG wire#powerrail
      I_Contact( #set_Motor )
      R_Coil( #CMD_A_Network_P4 )
   END_RUNG
   // the same network as SCL:
   IF NOT #set_Motor THEN #CMD_A_Network_P4 := FALSE; END_IF;
END_REGION
END_FUNCTION_BLOCK

FUNCTION "07_E_Correction PV HWrn LWrn" : Void
TITLE = Correction
{ S7_Optimized_Access := 'TRUE' }
AUTHOR : rtecmer
VERSION : 0.1
//Funkcja wprowadza korektę ostrzerzeń wysoki i niski poziom wartości procesowej. Wartości te są następnie wykorzystane podczas sterowania pompami dodatkowymi.
   VAR_INPUT 
      PV_HWrn_correction : Real;   // Wspóczninik służący wprowadzeniu korekty ostrzeżenia przekroczenia wartości zadanej bar
      PV_LWrn_correction : Real;   // Wspóczninik służący wprowadzeniu korekty ostrzeżenia zbyt niskia wartości bar w stosunku do zadanej
   END_VAR


BEGIN
	// Funkcja pozwala na wprowadzenie korekty sygnału ostrzeżenia
	// górnrgo i dolnego wartości procesowej
	
	
	
	
	//Przetwornik błąd górny
	"dbdane"."PID_Compact_1_sPid_Cmpt.r_Pv_Hlm" := "dbtags_Sterowanie".SetupControlPompownia.r_Pv_Hlm;
	"PID_Compact_1".sPid_Cmpt.r_Pv_Hlm := "dbdane"."PID_Compact_1_sPid_Cmpt.r_Pv_Hlm";
	
	//Przetwornik błąd dolny
	"dbdane"."PID_Compact_1_sPid_Cmpt.r_Pv_Llm" := "dbtags_Sterowanie".SetupControlPompownia.r_Pv_Llm;
	"PID_Compact_1".sPid_Cmpt.r_Pv_Llm := "dbdane"."PID_Compact_1_sPid_Cmpt.r_Pv_Llm";
	
	//***Wyliczenie ostrzerzeń HWrm i LWrm ***//
	IF "dbdane".Setpoint_SV <> 0 THEN
	  "dbdane"."PID_Compact_1_sPid_Cmpt.r_Pv_HWrn" := ("dbdane".Setpoint_SV + #PV_HWrn_correction);
	  "dbdane"."PID_Compact_1_sPid_Cmpt.r_Pv_LWrn" := ("dbdane".Setpoint_SV - #PV_LWrn_correction);
	  ;
	END_IF;
	
	
	
	//Ostrzegawczy wysoki
	"PID_Compact_1".sPid_Cmpt.r_Pv_HWrn := "dbdane"."PID_Compact_1_sPid_Cmpt.r_Pv_HWrn";
	"dbtags_Sterowanie".SetupControlPompownia.r_Pv_HWrn := "dbdane"."PID_Compact_1_sPid_Cmpt.r_Pv_HWrn";
	//Ostrzegawczy niski
	"PID_Compact_1".sPid_Cmpt.r_Pv_LWrn := "dbdane"."PID_Compact_1_sPid_Cmpt.r_Pv_LWrn";
	"dbtags_Sterowanie".SetupControlPompownia.r_Pv_LWrn := "dbdane"."PID_Compact_1_sPid_Cmpt.r_Pv_LWrn";
END_FUNCTION

FUNCTION_BLOCK "01_E_PID_Reset"   // FB6, LAD
TITLE = Reset regulator PID
{ S7_Optimized_Access := 'TRUE' }
AUTHOR : rtecmer
VERSION : 0.1
// Funkcja przeprowadza reset regulatora PID gdy utraci tryb automat czyli 3
// stored: AutoNumber true, IsIECCheckEnabled false, IsRetainMemResEnabled false, MemoryReserve 100, SetENOAutomatically false, UDAEnableTagReadback false
BEGIN

REGION Network 2: Histereza reset PID
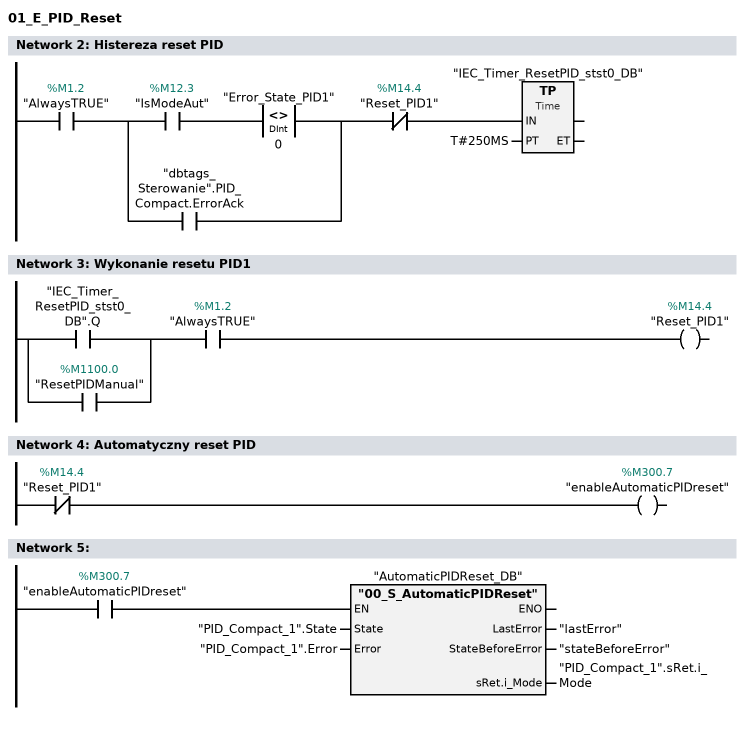
   RUNG wire#powerrail
      Contact( "AlwaysTRUE" )
      wire#w1
      Contact( "IsModeAut" )
      { S7_Templates := "SrcType := DInt" } NE_Contact(in1 := "Error_State_PID1", in2 := 0)
      wire#w2
      I_Contact( "Reset_PID1" )
      { S7_Templates := "time_type := Time" } "IEC_Timer_ResetPID_stst0_DB".TP(pt := T#250MS, et =>)
   END_RUNG
   RUNG wire#w1
      Contact( "dbtags_Sterowanie".PID_Compact.ErrorAck )
   END_RUNG wire#w2
   // the same network as SCL:
   "IEC_Timer_ResetPID_stst0_DB".TP(IN := "AlwaysTRUE" AND (("IsModeAut" AND ("Error_State_PID1" <> 0)) OR "dbtags_Sterowanie".PID_Compact.ErrorAck) AND NOT "Reset_PID1",
                           PT := T#250MS);
END_REGION

REGION Network 3: Wykonanie resetu PID1
   RUNG wire#powerrail
      Contact( "IEC_Timer_ResetPID_stst0_DB".Q )
      wire#w1
      Contact( "AlwaysTRUE" )
      Coil( "Reset_PID1" )
   END_RUNG
   RUNG wire#powerrail
      Contact( "ResetPIDManual" )
   END_RUNG wire#w1
   // the same network as SCL:
   "Reset_PID1" := ("IEC_Timer_ResetPID_stst0_DB".Q OR "ResetPIDManual") AND "AlwaysTRUE";
END_REGION

REGION Network 4: Automatyczny reset PID
   RUNG wire#powerrail
      I_Contact( "Reset_PID1" )
      Coil( "enableAutomaticPIDreset" )
   END_RUNG
   // the same network as SCL:
   "enableAutomaticPIDreset" := NOT "Reset_PID1";
END_REGION

REGION Network 5
   RUNG wire#powerrail
      Contact( "enableAutomaticPIDreset" )
      "AutomaticPIDReset_DB"(State := "PID_Compact_1".State, Error := "PID_Compact_1".Error, LastError => "lastError", StateBeforeError => "stateBeforeError", "sRet.i_Mode" => "PID_Compact_1".sRet.i_Mode)
   END_RUNG
   // the same network as SCL:
   IF "enableAutomaticPIDreset" THEN
       "AutomaticPIDReset_DB"(State := "PID_Compact_1".State,   // "00_S_AutomaticPIDReset"
                              Error := "PID_Compact_1".Error,
                              LastError => "lastError",
                              StateBeforeError => "stateBeforeError",
                              "sRet.i_Mode" => "PID_Compact_1".sRet.i_Mode);
   END_IF;
END_REGION
END_FUNCTION_BLOCK

FUNCTION_BLOCK "00_S_AutomaticPIDReset"   // FB22, LAD
{ S7_Optimized_Access := 'TRUE' }
VERSION : 0.1
// stored: AutoNumber true, IsIECCheckEnabled false, IsRetainMemResEnabled false, MemoryReserve 250, SetENOAutomatically false, UDAEnableTagReadback false
   VAR_INPUT
      State : Int;
      Error : DWord;
   END_VAR
   VAR_OUTPUT
      LastError : DWord;
      StateBeforeError : Int;
      "sRet.i_Mode" : Int;
   END_VAR
   VAR_TEMP   // added for the SCL form of the ladder/FBD networks
      _w1 : Bool;
   END_VAR
BEGIN

REGION Network 1: State Before Error
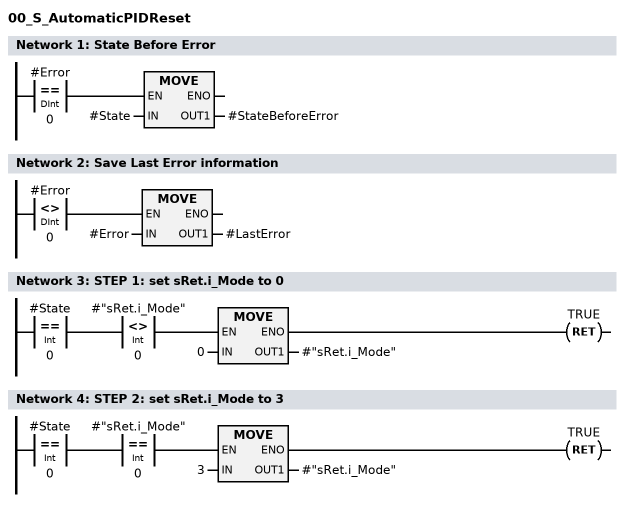
   RUNG wire#powerrail
      { S7_Templates := "SrcType := DInt" } EQ_Contact(in1 := #Error, in2 := 0)
      { S7_GenerateENO := "TRUE" } Move(in := #State, out1 => #StateBeforeError)
   END_RUNG
   // the same network as SCL:
   IF #Error = 0 THEN #StateBeforeError := #State; END_IF;
END_REGION

REGION Network 2: Save Last Error information
   RUNG wire#powerrail
      { S7_Templates := "SrcType := DInt" } NE_Contact(in1 := #Error, in2 := 0)
      { S7_GenerateENO := "TRUE" } Move(in := #Error, out1 => #LastError)
   END_RUNG
   // the same network as SCL:
   IF #Error <> 0 THEN #LastError := #Error; END_IF;
END_REGION

REGION Network 3: STEP 1: set sRet.i_Mode to 0
   // ENO of a box is taken as its EN; it also drops when the box reports an error
   #_w1 := (#State = 0) AND (#"sRet.i_Mode" <> 0);
   IF #_w1 THEN
       #"sRet.i_Mode" := 0;
       ENO := TRUE;
       RETURN;
   END_IF;
END_REGION

REGION Network 4: STEP 2: set sRet.i_Mode to 3
   // ENO of a box is taken as its EN; it also drops when the box reports an error
   #_w1 := (#State = 0) AND (#"sRet.i_Mode" = 0);
   IF #_w1 THEN
       #"sRet.i_Mode" := 3;
       ENO := TRUE;
       RETURN;
   END_IF;
END_REGION
END_FUNCTION_BLOCK

FUNCTION_BLOCK "04_A_Out_analog"   // FB23, LAD
TITLE = Output analogs
{ S7_Optimized_Access := 'TRUE' }
AUTHOR : rtecmer
VERSION : 0.1
// Obsługa wyjść analogowych
// stored: AutoNumber true, IsIECCheckEnabled false, IsRetainMemResEnabled false, MemoryReserve 100, SetENOAutomatically false, UDAEnableTagReadback false
   VAR
      Temp_SV_Int { ExternalAccessible := 'False'; ExternalVisible := 'False'; ExternalWritable := 'False'} : Int;
   END_VAR
   VAR_TEMP   // added for the SCL form of the ladder/FBD networks
      _w1 : Bool;
   END_VAR
BEGIN

REGION Network 1: Manual SV skalowanie
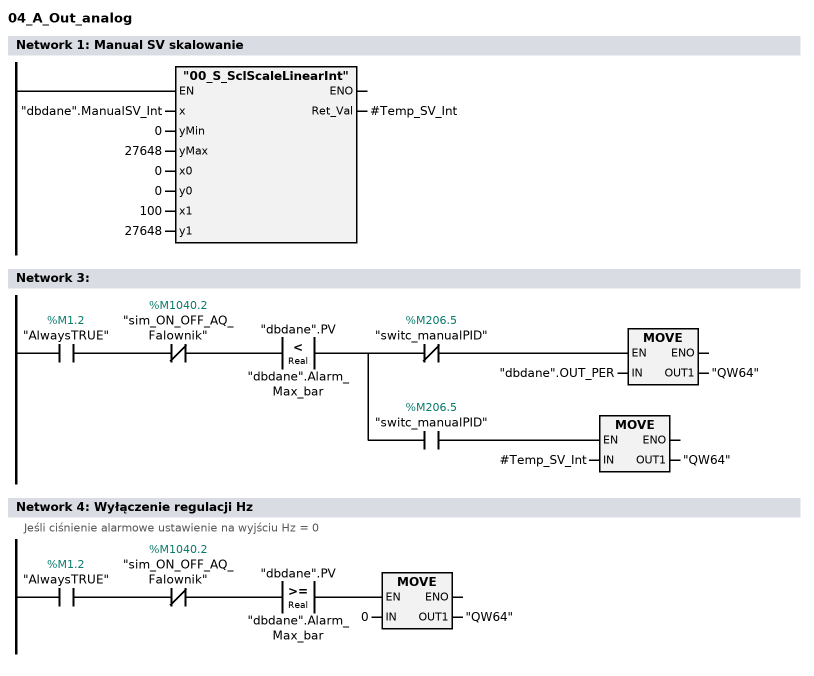
   RUNG wire#powerrail
      "00_S_SclScaleLinearInt"(x := "dbdane".ManualSV_Int, yMin := 0, yMax := 27648, x0 := 0, y0 := 0, x1 := 100, y1 := 27648, Ret_Val => #Temp_SV_Int)
   END_RUNG
   // the same network as SCL:
   #Temp_SV_Int := "00_S_SclScaleLinearInt"(x := "dbdane".ManualSV_Int,
                           yMin := 0,
                           yMax := 27648,
                           x0 := 0,
                           y0 := 0,
                           x1 := 100,
                           y1 := 27648);
END_REGION

REGION Network 3
   RUNG wire#powerrail
      Contact( "AlwaysTRUE" )
      I_Contact( "sim_ON_OFF_AQ_Falownik" )
      { S7_Templates := "SrcType := Real" } LT_Contact(in1 := "dbdane".PV, in2 := "dbdane".Alarm_Max_bar)
      wire#w1
      I_Contact( "switc_manualPID" )
      { S7_GenerateENO := "TRUE" } Move(in := "dbdane".OUT_PER, out1 => "QW64")
   END_RUNG
   RUNG wire#w1
      Contact( "switc_manualPID" )
      { S7_GenerateENO := "TRUE" } Move(in := #Temp_SV_Int, out1 => "QW64")
   END_RUNG
   // the same network as SCL:
   #_w1 := "AlwaysTRUE" AND NOT "sim_ON_OFF_AQ_Falownik" AND ("dbdane".PV < "dbdane".Alarm_Max_bar);
   IF #_w1 AND NOT "switc_manualPID" THEN "QW64" := "dbdane".OUT_PER; END_IF;
   IF #_w1 AND "switc_manualPID" THEN "QW64" := #Temp_SV_Int; END_IF;
END_REGION

REGION Network 4: Wyłączenie regulacji Hz
   // Jeśli ciśnienie alarmowe ustawienie na wyjściu Hz = 0
   RUNG wire#powerrail
      Contact( "AlwaysTRUE" )
      I_Contact( "sim_ON_OFF_AQ_Falownik" )
      { S7_Templates := "SrcType := Real" } GE_Contact(in1 := "dbdane".PV, in2 := "dbdane".Alarm_Max_bar)
      { S7_GenerateENO := "TRUE" } Move(in := 0, out1 => "QW64")
   END_RUNG
   // the same network as SCL:
   IF "AlwaysTRUE" AND NOT "sim_ON_OFF_AQ_Falownik" AND ("dbdane".PV >= "dbdane".Alarm_Max_bar) THEN
       "QW64" := 0;
   END_IF;
END_REGION
END_FUNCTION_BLOCK

FUNCTION "00_S_SclScaleLinearInt" : Int
{ S7_Optimized_Access := 'TRUE' }
VERSION : 0.1
   VAR_INPUT 
      x : Int;
      yMin : Int;   // Granica minimalnej wartości fizycznej
      yMax : Int;   // Granica maxymalnej wartości fizycznej
      x0 : Int;   // Minimalna wartość dla danego przetornika ADC zgodnie z dokumentacją Siemens
      y0 : Int;   // Minimalna wartość wartości fizycznej (procesowej)
      x1 : Int;   // Maxymalna wartość dla danego przetornika ADC zgodnie z dokumentacją Siemens
      y1 : Int;   // Maxymalna wartość wartości fizycznej (procesowej)
   END_VAR

   VAR_TEMP 
      tempYwert : Real;
      tempX0real : Real;
      tempX1real : Real;
      tempY0real : Real;
      tempY1real : Real;
      tempXreal : Real;
      tempYminReal : Real;
      tempYmaxReal : Real;
   END_VAR


BEGIN
	#tempX0real := INT_TO_REAL(#x0);
	#tempX1real := INT_TO_REAL(#x1);
	#tempY0real := INT_TO_REAL(#y0);
	#tempY1real := INT_TO_REAL(#y1);
	#tempXreal := INT_TO_REAL(#x);
	#tempYminReal := INT_TO_REAL(#yMin);
	#tempYmaxReal := INT_TO_REAL(#yMax);
	
	IF (#x1 - #x0) = 0 OR (#x - #x0) = 0 OR (#y1 - #y0) = 0 OR #yMin > #yMax
	THEN
	    #tempYwert := 0;
	ELSE
	    #tempYwert := (#tempY1real - #tempY0real) / (#tempX1real - #tempX0real) * (#tempXreal - #tempX0real) + #tempY0real;
	END_IF;
	
	IF #tempYwert < #tempYminReal THEN
	    #"00_S_SclScaleLinearInt" := 0;
	ELSIF #tempYwert > #tempYmaxReal THEN
	    #"00_S_SclScaleLinearInt" := #yMax;
	ELSE
	    #"00_S_SclScaleLinearInt" := REAL_TO_INT(#tempYwert);
	END_IF;
END_FUNCTION

FUNCTION "07_E_drivers pumps" : Void   // FC3, LAD
{ S7_Optimized_Access := 'TRUE' }
AUTHOR : RTecmer
VERSION : 0.1
// Sterowaniepompownią
// Funkcja zarządza sygnałem załączającym styczniki (sieć), (Falownik) danego napędu
// Sterowanie kompresorami
// Algorytm przewiduje sterowanie nadrzędne w trybie automatycznym przez sterownik master "OMROM". Sterowanie w trybie Manual z systemu SCADA odbywa się przez sterownik SLAVE "S7-1200" . Sterownik S7-100 reguluje sygnałem zadawania Hz w oparciu o regulator PID. Sygnał ten podawany jest na wejście analogowe sterownika Master. Praca sterownika S7-1200 Slave ogranicza się do generowania sygnału Hz, wystawianiu sygnału Automat, sygnału Dodatkowy kompresor 1, sygnału Dodatkowy kompresor 2. Komunikacji z systemem SCADA.
// stored: AutoNumber true, IsIECCheckEnabled false, SetENOAutomatically false, UDAEnableTagReadback false
BEGIN

REGION Network 1: Drive P1 / P1 Driver
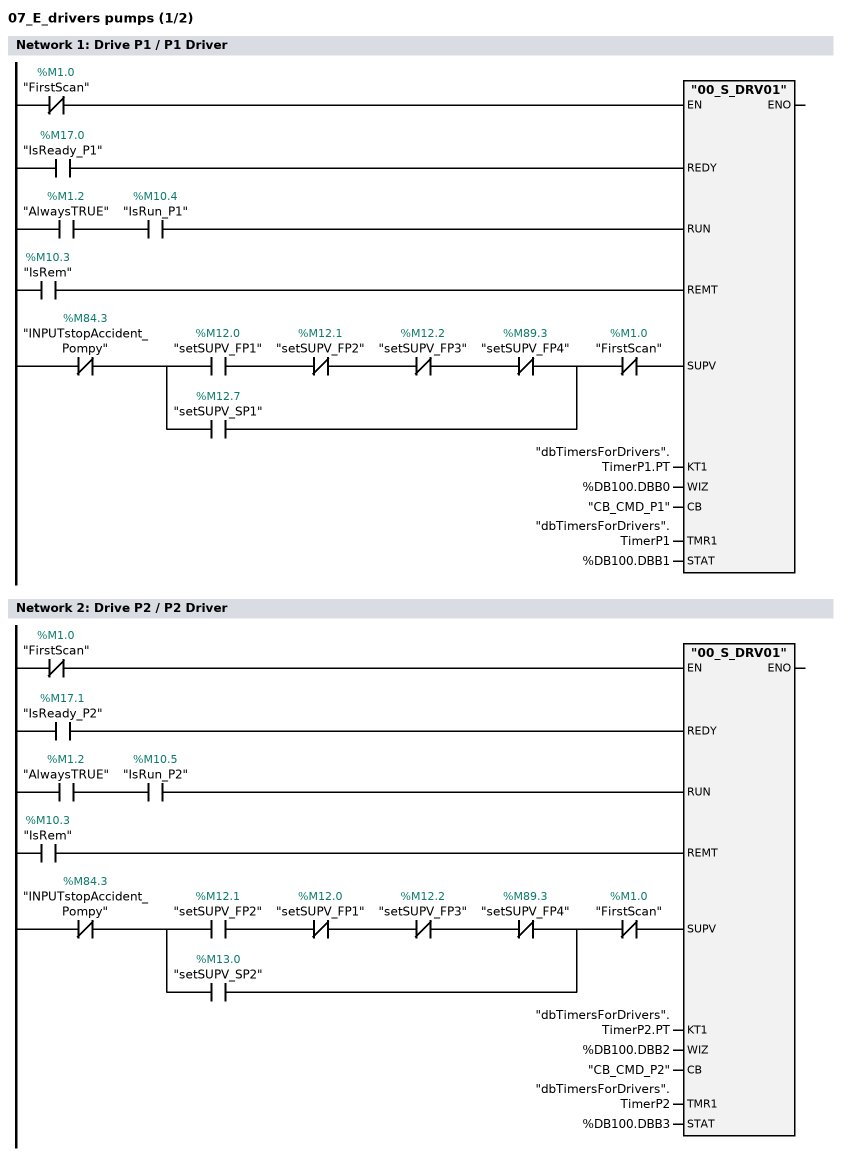
   RUNG wire#powerrail
      I_Contact( "FirstScan" )
      "00_S_DRV01"(REDY := wire#w1, RUN := wire#w2, REMT := wire#w3, SUPV := wire#w6, KT1 := "dbTimersForDrivers".TimerP1.PT, WIZ := %DB100.DBB0, CB := "CB_CMD_P1", TMR1 := "dbTimersForDrivers".TimerP1, STAT := %DB100.DBB1)
   END_RUNG
   RUNG wire#powerrail
      Contact( "IsReady_P1" )
   END_RUNG wire#w1
   RUNG wire#powerrail
      Contact( "AlwaysTRUE" )
      Contact( "IsRun_P1" )
   END_RUNG wire#w2
   RUNG wire#powerrail
      Contact( "IsRem" )
   END_RUNG wire#w3
   RUNG wire#powerrail
      I_Contact( "INPUTstopAccident_Pompy" )
      wire#w4
      Contact( "setSUPV_FP1" )
      I_Contact( "setSUPV_FP2" )
      I_Contact( "setSUPV_FP3" )
      I_Contact( "setSUPV_FP4" )
      wire#w5
      I_Contact( "FirstScan" )
   END_RUNG wire#w6
   RUNG wire#w4
      Contact( "setSUPV_SP1" )
   END_RUNG wire#w5
   // the same network as SCL:
   IF NOT "FirstScan" THEN
       "00_S_DRV01"(REDY := "IsReady_P1",
                    RUN := "AlwaysTRUE" AND "IsRun_P1",
                    REMT := "IsRem",
                    SUPV := NOT "INPUTstopAccident_Pompy" AND (("setSUPV_FP1" AND NOT "setSUPV_FP2" AND NOT "setSUPV_FP3" AND NOT "setSUPV_FP4") OR "setSUPV_SP1") AND NOT "FirstScan",
                    KT1 := "dbTimersForDrivers".TimerP1.PT,
                    WIZ := %DB100.DBB0,
                    CB := "CB_CMD_P1",
                    TMR1 := "dbTimersForDrivers".TimerP1,
                    STAT := %DB100.DBB1);
   END_IF;
END_REGION

REGION Network 2: Drive P2 / P2 Driver
   RUNG wire#powerrail
      I_Contact( "FirstScan" )
      "00_S_DRV01"(REDY := wire#w1, RUN := wire#w2, REMT := wire#w3, SUPV := wire#w6, KT1 := "dbTimersForDrivers".TimerP2.PT, WIZ := %DB100.DBB2, CB := "CB_CMD_P2", TMR1 := "dbTimersForDrivers".TimerP2, STAT := %DB100.DBB3)
   END_RUNG
   RUNG wire#powerrail
      Contact( "IsReady_P2" )
   END_RUNG wire#w1
   RUNG wire#powerrail
      Contact( "AlwaysTRUE" )
      Contact( "IsRun_P2" )
   END_RUNG wire#w2
   RUNG wire#powerrail
      Contact( "IsRem" )
   END_RUNG wire#w3
   RUNG wire#powerrail
      I_Contact( "INPUTstopAccident_Pompy" )
      wire#w4
      Contact( "setSUPV_FP2" )
      I_Contact( "setSUPV_FP1" )
      I_Contact( "setSUPV_FP3" )
      I_Contact( "setSUPV_FP4" )
      wire#w5
      I_Contact( "FirstScan" )
   END_RUNG wire#w6
   RUNG wire#w4
      Contact( "setSUPV_SP2" )
   END_RUNG wire#w5
   // the same network as SCL:
   IF NOT "FirstScan" THEN
       "00_S_DRV01"(REDY := "IsReady_P2",
                    RUN := "AlwaysTRUE" AND "IsRun_P2",
                    REMT := "IsRem",
                    SUPV := NOT "INPUTstopAccident_Pompy" AND (("setSUPV_FP2" AND NOT "setSUPV_FP1" AND NOT "setSUPV_FP3" AND NOT "setSUPV_FP4") OR "setSUPV_SP2") AND NOT "FirstScan",
                    KT1 := "dbTimersForDrivers".TimerP2.PT,
                    WIZ := %DB100.DBB2,
                    CB := "CB_CMD_P2",
                    TMR1 := "dbTimersForDrivers".TimerP2,
                    STAT := %DB100.DBB3);
   END_IF;
END_REGION

REGION Network 3: Drive P3 / P3 Driver
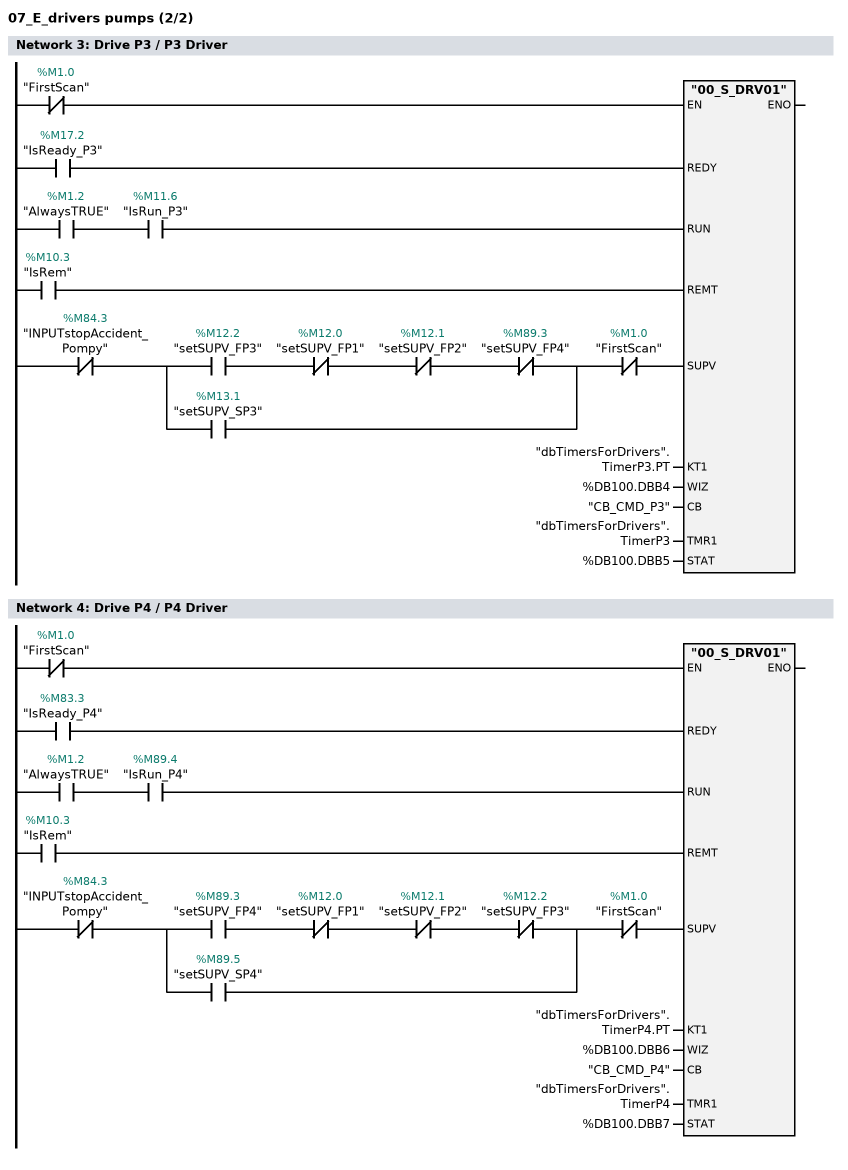
   RUNG wire#powerrail
      I_Contact( "FirstScan" )
      "00_S_DRV01"(REDY := wire#w1, RUN := wire#w2, REMT := wire#w3, SUPV := wire#w6, KT1 := "dbTimersForDrivers".TimerP3.PT, WIZ := %DB100.DBB4, CB := "CB_CMD_P3", TMR1 := "dbTimersForDrivers".TimerP3, STAT := %DB100.DBB5)
   END_RUNG
   RUNG wire#powerrail
      Contact( "IsReady_P3" )
   END_RUNG wire#w1
   RUNG wire#powerrail
      Contact( "AlwaysTRUE" )
      Contact( "IsRun_P3" )
   END_RUNG wire#w2
   RUNG wire#powerrail
      Contact( "IsRem" )
   END_RUNG wire#w3
   RUNG wire#powerrail
      I_Contact( "INPUTstopAccident_Pompy" )
      wire#w4
      Contact( "setSUPV_FP3" )
      I_Contact( "setSUPV_FP1" )
      I_Contact( "setSUPV_FP2" )
      I_Contact( "setSUPV_FP4" )
      wire#w5
      I_Contact( "FirstScan" )
   END_RUNG wire#w6
   RUNG wire#w4
      Contact( "setSUPV_SP3" )
   END_RUNG wire#w5
   // the same network as SCL:
   IF NOT "FirstScan" THEN
       "00_S_DRV01"(REDY := "IsReady_P3",
                    RUN := "AlwaysTRUE" AND "IsRun_P3",
                    REMT := "IsRem",
                    SUPV := NOT "INPUTstopAccident_Pompy" AND (("setSUPV_FP3" AND NOT "setSUPV_FP1" AND NOT "setSUPV_FP2" AND NOT "setSUPV_FP4") OR "setSUPV_SP3") AND NOT "FirstScan",
                    KT1 := "dbTimersForDrivers".TimerP3.PT,
                    WIZ := %DB100.DBB4,
                    CB := "CB_CMD_P3",
                    TMR1 := "dbTimersForDrivers".TimerP3,
                    STAT := %DB100.DBB5);
   END_IF;
END_REGION

REGION Network 4: Drive P4 / P4 Driver
   RUNG wire#powerrail
      I_Contact( "FirstScan" )
      "00_S_DRV01"(REDY := wire#w1, RUN := wire#w2, REMT := wire#w3, SUPV := wire#w6, KT1 := "dbTimersForDrivers".TimerP4.PT, WIZ := %DB100.DBB6, CB := "CB_CMD_P4", TMR1 := "dbTimersForDrivers".TimerP4, STAT := %DB100.DBB7)
   END_RUNG
   RUNG wire#powerrail
      Contact( "IsReady_P4" )
   END_RUNG wire#w1
   RUNG wire#powerrail
      Contact( "AlwaysTRUE" )
      Contact( "IsRun_P4" )
   END_RUNG wire#w2
   RUNG wire#powerrail
      Contact( "IsRem" )
   END_RUNG wire#w3
   RUNG wire#powerrail
      I_Contact( "INPUTstopAccident_Pompy" )
      wire#w4
      Contact( "setSUPV_FP4" )
      I_Contact( "setSUPV_FP1" )
      I_Contact( "setSUPV_FP2" )
      I_Contact( "setSUPV_FP3" )
      wire#w5
      I_Contact( "FirstScan" )
   END_RUNG wire#w6
   RUNG wire#w4
      Contact( "setSUPV_SP4" )
   END_RUNG wire#w5
   // the same network as SCL:
   IF NOT "FirstScan" THEN
       "00_S_DRV01"(REDY := "IsReady_P4",
                    RUN := "AlwaysTRUE" AND "IsRun_P4",
                    REMT := "IsRem",
                    SUPV := NOT "INPUTstopAccident_Pompy" AND (("setSUPV_FP4" AND NOT "setSUPV_FP1" AND NOT "setSUPV_FP2" AND NOT "setSUPV_FP3") OR "setSUPV_SP4") AND NOT "FirstScan",
                    KT1 := "dbTimersForDrivers".TimerP4.PT,
                    WIZ := %DB100.DBB6,
                    CB := "CB_CMD_P4",
                    TMR1 := "dbTimersForDrivers".TimerP4,
                    STAT := %DB100.DBB7);
   END_IF;
END_REGION
END_FUNCTION

FUNCTION "00_S_DRV01" : Void   // FC1, LAD
TITLE = Funkcja sterowania stycznikiem silnika
{ S7_Optimized_Access := 'FALSE' }
VERSION : 0.1
// Funkcja standardowa sluzy do zalaczania silnika.
// Posiada trzy tryby pracy:
//      - localny (zalaczanie  elektrycznie bez PLC)
//      - zdalny  (zalaczanie przez PLC)
//          - reczny (zalaczanie przez dyspozytora z SCADA)
//          - automatyczny (zalaczanie wynikle z algotytmu sterowania)
// Zrodlo danych dla funkcji stanowia:
//      - sygnaly I/O PLC
//          - =REDY -gotowosc napedu
//          - =REMT -sterowanie napedu 1-zdalnie 0-local
//          - =RUN  -naped wlaczony
//          - =CB   -zalaczenie stycznika
//       - =STAT bajt statusu napedu 
//               jego kopia w DB =WIZ stanowi interface PLC/MMI
//          - bit 0 Alarm              (sygnal do MMI)
//          - bit 1  
//          - bit 2 kopia sygnalu REMT (sygnal do SCADA)
//          - bit 3 kopia sygnalu RUN  (sygnal do SCADA)
//          - bit 4 wylaczenie reczne  (sygnal z SCADA) 
//          - bit 5 wlaczenie reczne   (sygnal z SCADA)
//          - bit 6 alarm reset        (sygnal z SCADA)
//          - bit 7 1=auto, 0=man      (sygnal z SCADA)
//        - =SUPV - sygnal zalacznia w trybie automatycznym
//        - sygnaly czasowe
//          - =TMR1 -kontrola czasu zalaczenia stycznika
//          - =KT1  -wartosc czasu timera 1
//          - flagi
// stored: AutoNumber false, IsIECCheckEnabled false, SetENOAutomatically false, UDAEnableTagReadback false
   VAR_INPUT
      REDY : Bool;   // Sygnał gotowości
      RUN : Bool;   // Sygnał pracy
      REMT : Bool;   // Sterowanie napędu zdalne-1 lokalne -0
      SUPV : Bool;   // Sygnalizacja załączenia w trybie automatycznym
      KT1 : Time;   // wartosc czasu timera 1
   END_VAR
   VAR_IN_OUT
      WIZ : Byte;   // Wektor stanu ze SCADA
      CB : Bool;   // Przekaźnik urządzenia
      TMR1 : TON_TIME;   // Kontrola czasu załączenia stycznika
      STAT : Byte;   // Wektor stanu urządzenia
   END_VAR
   // Ret_Val : Napęd jednokierunkowy - pompy
BEGIN

REGION Network 1: Network 1: mapowanie wektora statusu napędu i stanu wektora z SCADA
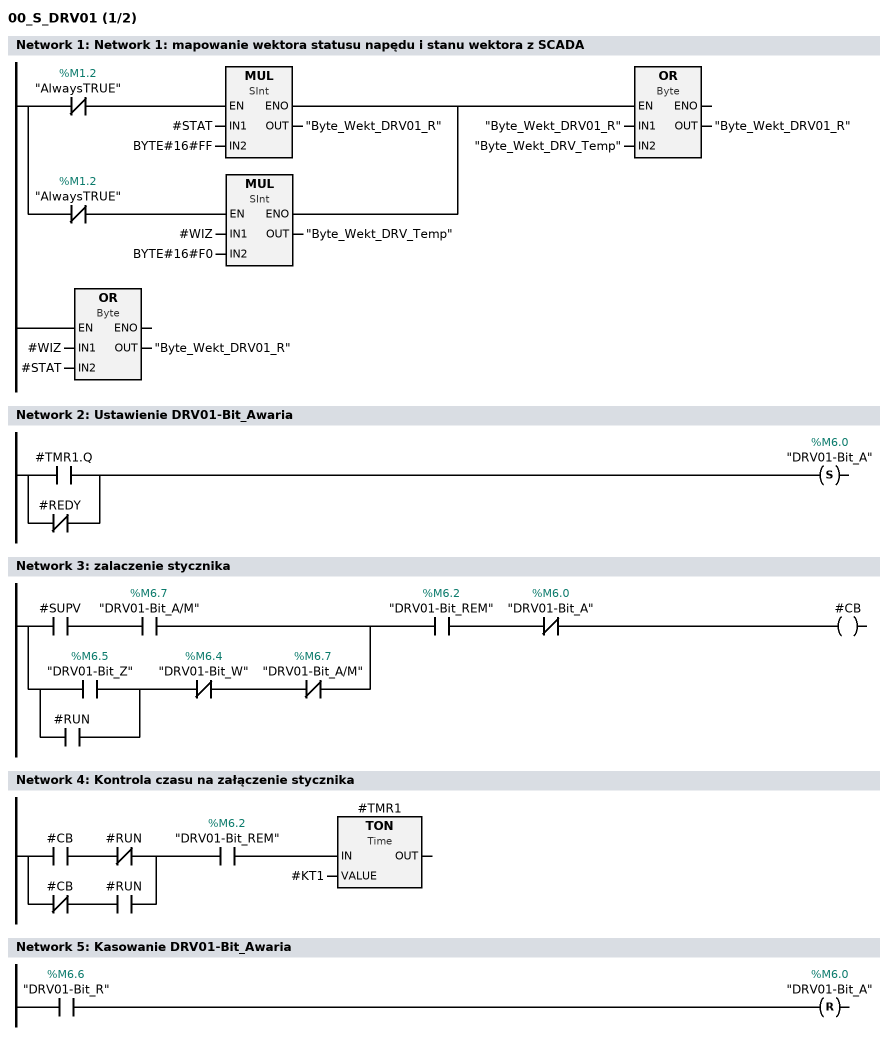
   // ENO of a box is taken as its EN; it also drops when the box reports an error
   IF NOT "AlwaysTRUE" THEN
       "Byte_Wekt_DRV01_R" := #STAT * BYTE#16#FF;
       "Byte_Wekt_DRV_Temp" := #WIZ * BYTE#16#F0;
   END_IF;
   IF NOT "AlwaysTRUE" OR NOT "AlwaysTRUE" THEN
       "Byte_Wekt_DRV01_R" := "Byte_Wekt_DRV01_R" OR "Byte_Wekt_DRV_Temp";
   END_IF;
   "Byte_Wekt_DRV01_R" := #WIZ OR #STAT;
END_REGION

REGION Network 2: Ustawienie DRV01-Bit_Awaria
   RUNG wire#powerrail
      Contact( #TMR1.Q )
      wire#w1
      S_Coil( "DRV01-Bit_A" )
   END_RUNG
   RUNG wire#powerrail
      I_Contact( #REDY )
   END_RUNG wire#w1
   // the same network as SCL:
   IF #TMR1.Q OR NOT #REDY THEN "DRV01-Bit_A" := TRUE; END_IF;
END_REGION

REGION Network 3: zalaczenie stycznika
   RUNG wire#powerrail
      Contact( #SUPV )
      Contact( "DRV01-Bit_A/M" )
      wire#w1
      Contact( "DRV01-Bit_REM" )
      I_Contact( "DRV01-Bit_A" )
      Coil( #CB )
   END_RUNG
   RUNG wire#powerrail
      Contact( "DRV01-Bit_Z" )
      wire#w2
      I_Contact( "DRV01-Bit_W" )
      I_Contact( "DRV01-Bit_A/M" )
   END_RUNG wire#w1
   RUNG wire#powerrail
      Contact( #RUN )
   END_RUNG wire#w2
   // the same network as SCL:
   #CB := ((#SUPV AND "DRV01-Bit_A/M") OR (("DRV01-Bit_Z" OR #RUN) AND NOT "DRV01-Bit_W" AND NOT "DRV01-Bit_A/M")) AND "DRV01-Bit_REM" AND NOT "DRV01-Bit_A";
END_REGION

REGION Network 4: Kontrola czasu na załączenie stycznika
   #TMR1(IN := ((#CB AND NOT #RUN) OR (NOT #CB AND #RUN)) AND "DRV01-Bit_REM", PT := #KT1);   // TON coil
END_REGION

REGION Network 5: Kasowanie DRV01-Bit_Awaria
   RUNG wire#powerrail
      Contact( "DRV01-Bit_R" )
      R_Coil( "DRV01-Bit_A" )
   END_RUNG
   // the same network as SCL:
   IF "DRV01-Bit_R" THEN "DRV01-Bit_A" := FALSE; END_IF;
END_REGION

REGION Network 6: Bit Out wektora napędu sygnał Alarm
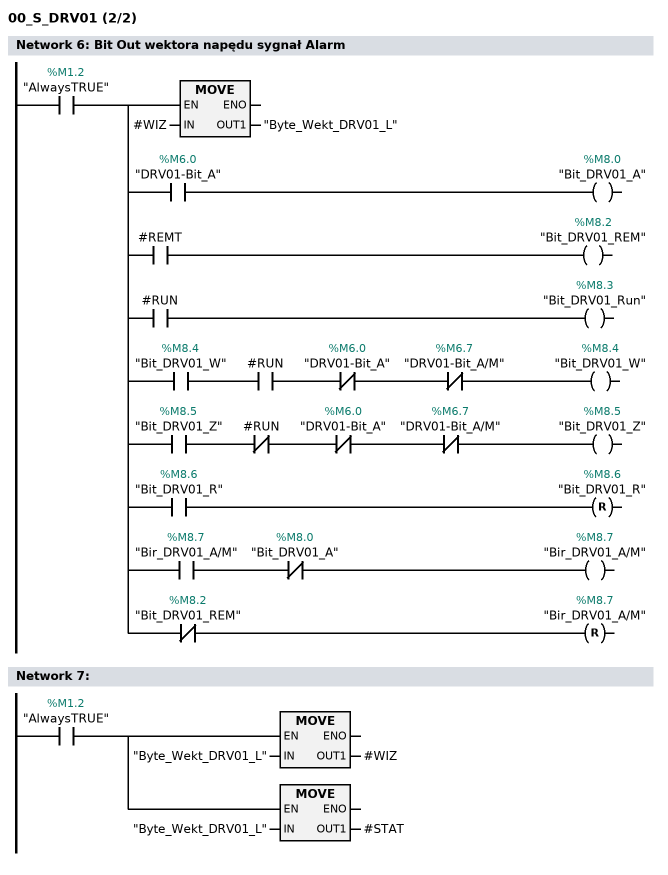
   RUNG wire#powerrail
      Contact( "AlwaysTRUE" )
      wire#w1
      { S7_GenerateENO := "TRUE" } Move(in := #WIZ, out1 => "Byte_Wekt_DRV01_L")
   END_RUNG
   RUNG wire#w1
      Contact( "DRV01-Bit_A" )
      Coil( "Bit_DRV01_A" )
   END_RUNG
   RUNG wire#w1
      Contact( #REMT )
      Coil( "Bit_DRV01_REM" )
   END_RUNG
   RUNG wire#w1
      Contact( #RUN )
      Coil( "Bit_DRV01_Run" )
   END_RUNG
   RUNG wire#w1
      Contact( "Bit_DRV01_W" )
      Contact( #RUN )
      I_Contact( "DRV01-Bit_A" )
      I_Contact( "DRV01-Bit_A/M" )
      Coil( "Bit_DRV01_W" )
   END_RUNG
   RUNG wire#w1
      Contact( "Bit_DRV01_Z" )
      I_Contact( #RUN )
      I_Contact( "DRV01-Bit_A" )
      I_Contact( "DRV01-Bit_A/M" )
      Coil( "Bit_DRV01_Z" )
   END_RUNG
   RUNG wire#w1
      Contact( "Bit_DRV01_R" )
      R_Coil( "Bit_DRV01_R" )
   END_RUNG
   RUNG wire#w1
      Contact( "Bir_DRV01_A/M" )
      I_Contact( "Bit_DRV01_A" )
      Coil( "Bir_DRV01_A/M" )
   END_RUNG
   RUNG wire#w1
      I_Contact( "Bit_DRV01_REM" )
      R_Coil( "Bir_DRV01_A/M" )
   END_RUNG
   // the same network as SCL:
   IF "AlwaysTRUE" THEN "Byte_Wekt_DRV01_L" := #WIZ; END_IF;
   "Bit_DRV01_A" := "AlwaysTRUE" AND "DRV01-Bit_A";
   "Bit_DRV01_REM" := "AlwaysTRUE" AND #REMT;
   "Bit_DRV01_Run" := "AlwaysTRUE" AND #RUN;
   "Bit_DRV01_W" := "AlwaysTRUE" AND "Bit_DRV01_W" AND #RUN AND NOT "DRV01-Bit_A" AND NOT "DRV01-Bit_A/M";
   "Bit_DRV01_Z" := "AlwaysTRUE" AND "Bit_DRV01_Z" AND NOT #RUN AND NOT "DRV01-Bit_A" AND NOT "DRV01-Bit_A/M";
   IF "AlwaysTRUE" AND "Bit_DRV01_R" THEN "Bit_DRV01_R" := FALSE; END_IF;
   "Bir_DRV01_A/M" := "AlwaysTRUE" AND "Bir_DRV01_A/M" AND NOT "Bit_DRV01_A";
   IF "AlwaysTRUE" AND NOT "Bit_DRV01_REM" THEN "Bir_DRV01_A/M" := FALSE; END_IF;
END_REGION

REGION Network 7
   RUNG wire#powerrail
      Contact( "AlwaysTRUE" )
      wire#w1
      { S7_GenerateENO := "TRUE" } Move(in := "Byte_Wekt_DRV01_L", out1 => #WIZ)
   END_RUNG
   RUNG wire#w1
      { S7_GenerateENO := "TRUE" } Move(in := "Byte_Wekt_DRV01_L", out1 => #STAT)
   END_RUNG
   // the same network as SCL:
   IF "AlwaysTRUE" THEN
       #WIZ := "Byte_Wekt_DRV01_L";
       #STAT := "Byte_Wekt_DRV01_L";
   END_IF;
END_REGION
END_FUNCTION

FUNCTION "07_E_Commutation of Contactors" : Void
TITLE = Blok sterowania stycznikami F/S i sygnał ON/OFF Soft-Start/ Falo
{ S7_Optimized_Access := 'TRUE' }
AUTHOR : rtecmer
VERSION : 0.1
//Funkcja służy do sterowania stycznikami sieć, falownik napędów P1-P4. 

BEGIN
	(*
	//=============================================================================
	//(JZWiK S.A Radosław Tecmer)
	//(c)Copyright (2021) All Rights Reserved
	//-----------------------------------------------------------------------------
	//Testowane z:   (system docelowy z  FW 4.4)
	//Pakiet inżynierski:   TIA Portal (V14 Sp1 Update 9)
	//Ograniczenia:  ( - )
	//Wymagania:  (minimalne S7-1200 CPU 1215C FW 4.2 .)
	//Funkcjonalnośc: (Komutacja styczników F/S. Sterowanie sygnałami On/Off soft-start
	//                i falownik)
	//-----------------------------------------------------------------------------
	//Zmainy wprowadzone:
	//Wersja  Data       Osoba wprowadzająca zmiany - ekspert
	//01.00.00 09.1.2022 (Tecmer Radosław - twórca) Pieresza wersja 01.00.00
	//=============================================================================
	*)
	
	
	
	REGION Pompa P1 
	  // sterowanie stycznikami falownik
	  IF ("CB_CMD_P1" = 1)AND ("IsReady_Inverter"=1) AND ("IsReady_P1" = 1) AND NOT "IsCurrentOverloadInverter" AND
	    ("setCMD_FP1" = 1) AND
	    ("CMD_network_P1" = 0) AND
	    ("CMD_inverter_P2" = 0) AND ("CMD_inverter_P3" = 0) AND ("CMD_inverter_P4" = 0)
	  THEN
	    // Sterowanie stycznikiem falownika 
	    "CMD_inverter_P1" := TRUE;
	  ELSE
	    "CMD_inverter_P1" := FALSE;
	    ;
	  END_IF;
	  
	
	  
	  // Sterowanie stycznikiem sieć 
	  // sterowanie automat
	  IF (("CB_CMD_P1" = 1) AND ("IsReady_P1" = 1) AND
	    ("setCMD_SP1" = 1) AND
	    ("CMD_inverter_P1" = 0))
	    OR
	    ("CB_CMD_P1" = 1 AND "bitH_Aut_Man_P1" = 0 AND "CMD_inverter_P1" = 0) // sterowanie manual
	  THEN
	    // Sterowanie stycznikiem sieć 
	    "CMD_network_P1" := TRUE;
	  ELSE
	    "CMD_network_P1" := FALSE;
	    ;
	  END_IF;
	  
	 
	  (*
	  // Sterowanie sygnałem podawanym na Soft-Start
	  IF "inputRunS_P1" AND "IsReady_P1" = TRUE AND"IsRem" THEN
	    // Podaj sybnał start na soft-start
	    "CMD_soft_P1" := "inputRunS_P1";
	  ELSE
	    "CMD_soft_P1" := FALSE;
	    ;
	  END_IF;
	  *)
	  
	  
	END_REGION
	
	REGION Pompa P2
	  // sterowanie stycznikami falownik
	  IF ("CB_CMD_P2" = 1)AND ("IsReady_Inverter"=1) AND ("IsReady_P2" = 1) AND NOT "IsCurrentOverloadInverter" AND
	    ("setCMD_FP2" = 1) AND
	    ("CMD_network_P2" = 0) AND
	    ("CMD_inverter_P1" = 0) AND ("CMD_inverter_P3" = 0) AND ("CMD_inverter_P4" = 0)
	    
	  THEN
	    // Sterowanie stycznikiem falownika
	    "CMD_inverter_P2" := TRUE;
	  ELSE
	    "CMD_inverter_P2" := FALSE;
	    ;
	  END_IF;
	  
	
	  
	  // Sterowanie stycznikiem sieć 
	  // sterowanie automat
	  IF (("CB_CMD_P2" = 1) AND ("IsReady_P2" = 1) AND
	    ("setCMD_SP2" = 1) AND
	    ("CMD_inverter_P2" = 0))
	    OR
	    ("CB_CMD_P2" = 1 AND "bitH_Aut_Man_P2" = 0 AND "CMD_inverter_P2" = 0 ) // sterowanie manual
	  THEN
	    // Sterowanie stycznikiem sieć 
	    "CMD_network_P2" := TRUE;
	  ELSE
	    "CMD_network_P2" := FALSE;
	    ;
	  END_IF;
	  
	 
	  (*
	  // Sterowanie sygnałem podawanym na Soft-Start
	  IF "inputRunS_P2" AND "IsReady_P2" = TRUE AND  "IsRem" THEN
	    // Podaj sybnał start na soft-start
	    "CMD_soft_P2" := "inputRunS_P2";
	  ELSE
	    "CMD_soft_P2" := FALSE;
	    ;
	  END_IF;
	  *)
	  
	END_REGION
	
	REGION Pompa P3
	  // sterowanie stycznikami falownik
	  IF ("CB_CMD_P3" = 1)AND ("IsReady_Inverter"=1) AND ("IsReady_P3" = 1) AND NOT "IsCurrentOverloadInverter" AND
	    ("setCMD_FP3" = 1) AND
	    ("CMD_network_P3" = 0) AND
	    ("CMD_inverter_P2" = 0) AND ("CMD_inverter_P1" = 0) AND ("CMD_inverter_P4" = 0) 
	  THEN
	    // Sterowanie stycznikiem falownika 
	    "CMD_inverter_P3" := TRUE;
	  ELSE
	    "CMD_inverter_P3" := FALSE;
	    ;
	  END_IF;
	  
	 
	  
	  // Sterowanie stycznikiem sieć 
	  // sterowanie automt
	  IF (("CB_CMD_P3" = 1) AND ("IsReady_P3" = 1) AND
	    ("setCMD_SP3" = 1) AND
	    ("CMD_inverter_P3" = 0))
	    OR
	    ("CB_CMD_P3" = 1 AND "bitH_Aut_Man_P3" = 0 AND "CMD_inverter_P3" = 0) // sterowanie manual
	  THEN
	     //Sterowanie stycznikiem sieć 
	    "CMD_network_P3" := TRUE;
	  ELSE
	    "CMD_network_P3" := FALSE;
	    ;
	  END_IF;
	  
	 
	  (*
	  // Sterowanie sygnałem podawanym na Soft-Start
	  IF "inputRunS_P3" AND "IsReady_P3"= TRUE AND  "IsRem" THEN
	     //Podaj sybnał start na soft-start
	    "CMD_soft_P3" := "inputRunS_P3";
	  ELSE
	    "CMD_soft_P3":= FALSE;
	    ;
	  END_IF;
	  *)
	  
	END_REGION
	
	
	
	REGION Pompa P4
	  // sterowanie stycznikami falownik
	  IF ("CB_CMD_P4" = 1)AND ("IsReady_Inverter"=1) AND ("IsReady_P4" = 1) AND NOT "IsCurrentOverloadInverter" AND
	    ("setCMD_FP4" = 1) AND
	    ("CMD_network_P4" = 0) AND
	    ("CMD_inverter_P2" = 0) AND ("CMD_inverter_P1" = 0) AND ("CMD_inverter_P3" = 0)
	  THEN
	    // Sterowanie stycznikiem falownika 
	    "CMD_inverter_P4" := TRUE;
	  ELSE
	    "CMD_inverter_P4" := FALSE;
	    ;
	  END_IF;
	  
	       // Sterowanie stycznikiem sieć 
	      // sterowanie automaat 
	  IF (("CB_CMD_P4" = 1) AND ("IsReady_P4" = 1) AND
	    ("setCMD_SP4" = 1) AND
	    ("CMD_inverter_P4" = 0))
	    OR
	    ("CB_CMD_P4" = 1 AND "bitH_Aut_Man_P4" = 0 AND "CMD_inverter_P4" = 0) // sterowanie manual
	  THEN
	    // Sterowanie stycznikiem sieć 
	    "CMD_network_P4" := TRUE;
	  ELSE
	    "CMD_network_P4" := FALSE;
	    ;
	  END_IF;
	  
	
	  
	  (*
	  // Sterowanie sygnałem podawanym na Soft-Start
	  IF "inputRunS_P4" AND "IsReady_P4"= TRUE AND  "IsRem" THEN
	    // Podaj sybnał start na soft-start
	    "CMD_soft_P4" := "inputRunS_P4" ;
	  ELSE
	    "CMD_soft_P4" := FALSE;
	    ;
	  END_IF;
	  *)
	  
	END_REGION
END_FUNCTION

FUNCTION "00_S_Reset" : Void   // FC7, LAD
TITLE = Reset PID
{ S7_Optimized_Access := 'TRUE' }
AUTHOR : RTecmer
VERSION : 0.1
// (*
// //=============================================================================
// //(JZWiK S.A Radosław Tecmer)
// //(c)Copyright (2021) All Rights Reserved
// //-----------------------------------------------------------------------------
// //Testowane z:   (system docelowy z  FW 4.4)
// //Pakiet inżynierski:   TIA Portal (V14 Sp1 Update 9)
// //Ograniczenia:  ( - )
// //Wymagania:  (minimalne S7-1200 CPU 1215C FW 4.2 .)
// //Funkcjonalnośc: (Reset błędu i ustawienie wartości domyślnych PID )
// //-----------------------------------------------------------------------------
// //Zmainy wprowadzone:
// //Wersja  Data       Osoba wprowadzająca zmiany - ekspert
// //01.00.00 17.11.2021 (Tecmer Radosław - twórca) Pieresza wersja 01.00.00
// //=============================================================================
// *)
// stored: AutoNumber true, IsIECCheckEnabled false, SetENOAutomatically false, UDAEnableTagReadback false
BEGIN
END_FUNCTION

FUNCTION "04_A_Convert_Scaling_analog" : Void   // FC14, LAD
TITLE = Funkcja konwertera analogów
{ S7_Optimized_Access := 'TRUE' }
AUTHOR : RTecmer
VERSION : 0.1
// Konwertowanie zmiennych procesowych
// stored: AutoNumber true, IsIECCheckEnabled false, SetENOAutomatically false, UDAEnableTagReadback false
BEGIN

REGION Network 1: Przepywomierz Q1 Pompownia
   // Pobrane z Modbus RTU
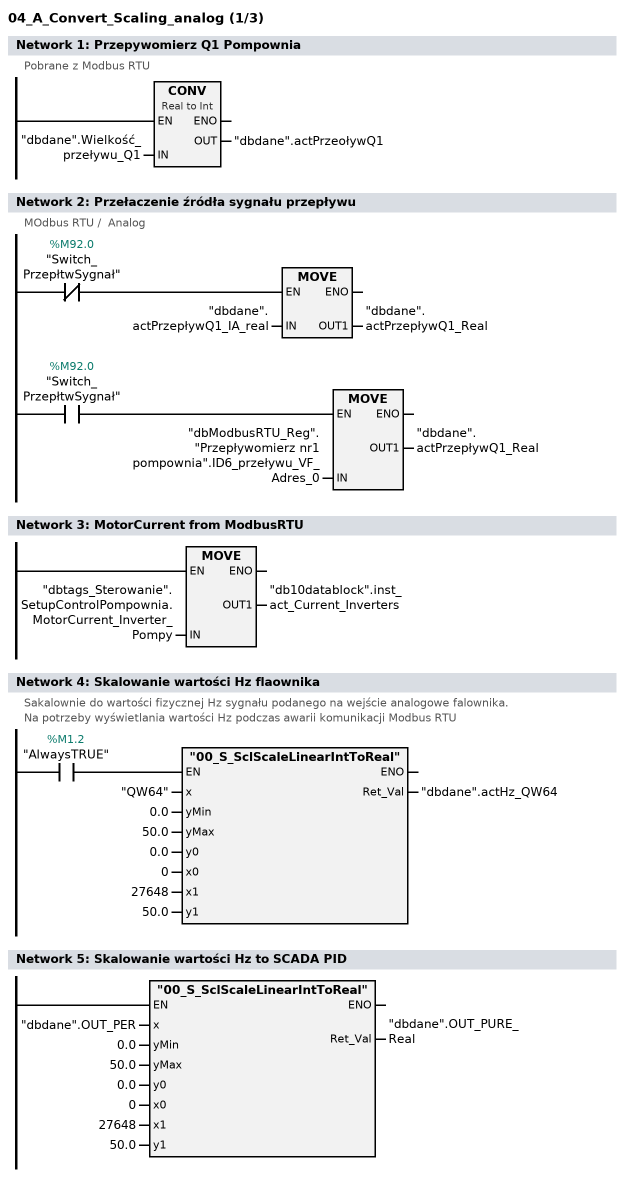
   RUNG wire#powerrail
      { S7_Templates := "[SrcType := Real, DestType := Int]" } Convert(in := "dbdane".Wielkość_przeływu_Q1, out => "dbdane".actPrzeoływQ1)
   END_RUNG
   // the same network as SCL:
   "dbdane".actPrzeoływQ1 := REAL_TO_INT("dbdane".Wielkość_przeływu_Q1);
END_REGION

REGION Network 2: Przełaczenie źródła sygnału przepływu
   // MOdbus RTU /  Analog
   RUNG wire#powerrail
      I_Contact( "Switch_PrzepłtwSygnał" )
      Move(in := "dbdane".actPrzepływQ1_IA_real, out1 => "dbdane".actPrzepływQ1_Real)
   END_RUNG
   RUNG wire#powerrail
      Contact( "Switch_PrzepłtwSygnał" )
      Move(in := "dbModbusRTU_Reg"."Przepływomierz nr1 pompownia".ID6_przeływu_VF_Adres_0, out1 => "dbdane".actPrzepływQ1_Real)
   END_RUNG
   // the same network as SCL:
   IF NOT "Switch_PrzepłtwSygnał" THEN "dbdane".actPrzepływQ1_Real := "dbdane".actPrzepływQ1_IA_real; END_IF;
   IF "Switch_PrzepłtwSygnał" THEN
       "dbdane".actPrzepływQ1_Real := "dbModbusRTU_Reg"."Przepływomierz nr1 pompownia".ID6_przeływu_VF_Adres_0;
   END_IF;
END_REGION

REGION Network 3: MotorCurrent from ModbusRTU
   RUNG wire#powerrail
      Move(in := "dbtags_Sterowanie".SetupControlPompownia.MotorCurrent_Inverter_Pompy, out1 => "db10datablock".inst_act_Current_Inverters)
   END_RUNG
   // the same network as SCL:
   "db10datablock".inst_act_Current_Inverters := "dbtags_Sterowanie".SetupControlPompownia.MotorCurrent_Inverter_Pompy;
END_REGION

REGION Network 4: Skalowanie wartości Hz flaownika
   // Sakalownie do wartości fizycznej Hz sygnału podanego na wejście analogowe falownika.
   // Na potrzeby wyświetlania wartości Hz podczas awarii komunikacji Modbus RTU
   RUNG wire#powerrail
      Contact( "AlwaysTRUE" )
      "00_S_SclScaleLinearIntToReal"(x := "QW64", yMin := 0.0, yMax := 50.0, y0 := 0.0, x0 := 0, x1 := 27648, y1 := 50.0, Ret_Val => "dbdane".actHz_QW64)
   END_RUNG
   // the same network as SCL:
   IF "AlwaysTRUE" THEN
       "dbdane".actHz_QW64 := "00_S_SclScaleLinearIntToReal"(x := "QW64",
                               yMin := 0.0,
                               yMax := 50.0,
                               y0 := 0.0,
                               x0 := 0,
                               x1 := 27648,
                               y1 := 50.0);
   END_IF;
END_REGION

REGION Network 5: Skalowanie wartości Hz to SCADA PID
   RUNG wire#powerrail
      "00_S_SclScaleLinearIntToReal"(x := "dbdane".OUT_PER, yMin := 0.0, yMax := 50.0, y0 := 0.0, x0 := 0, x1 := 27648, y1 := 50.0, Ret_Val => "dbdane".OUT_PURE_Real)
   END_RUNG
   // the same network as SCL:
   "dbdane".OUT_PURE_Real := "00_S_SclScaleLinearIntToReal"(x := "dbdane".OUT_PER,
                           yMin := 0.0,
                           yMax := 50.0,
                           y0 := 0.0,
                           x0 := 0,
                           x1 := 27648,
                           y1 := 50.0);
END_REGION

REGION Network 7: Ciśnienie kierunek miasto
   // Pomiar z czujnika B6 poziom "Przetłaczanie" - wylot za zasuwą
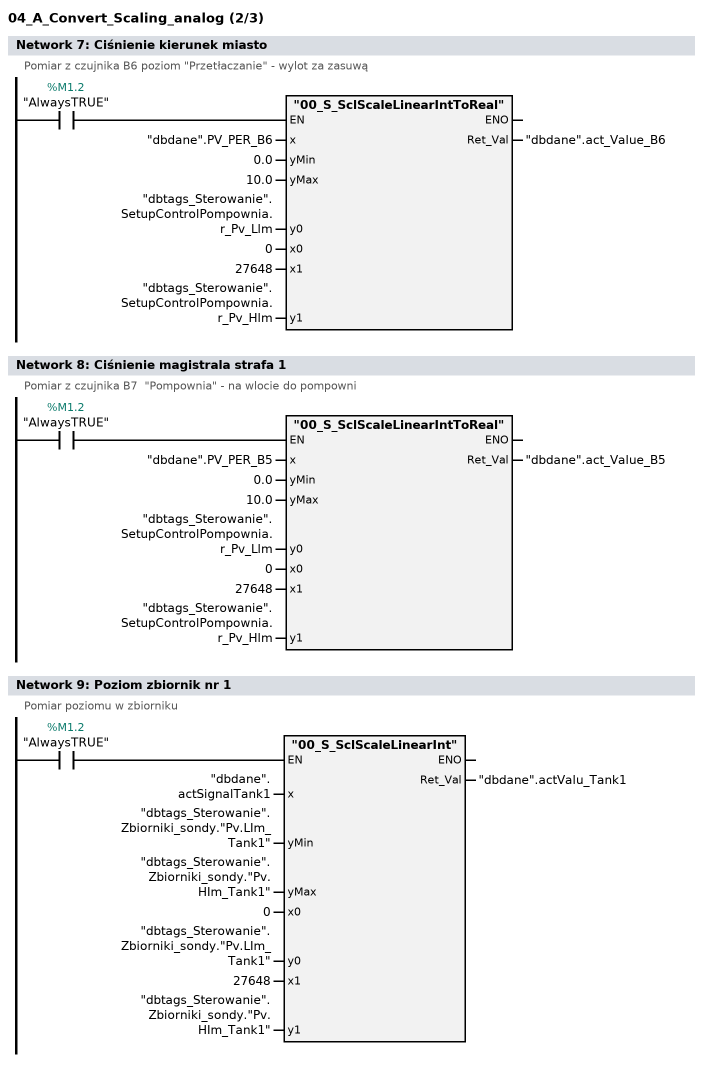
   RUNG wire#powerrail
      Contact( "AlwaysTRUE" )
      "00_S_SclScaleLinearIntToReal"(x := "dbdane".PV_PER_B6, yMin := 0.0, yMax := 10.0, y0 := "dbtags_Sterowanie".SetupControlPompownia.r_Pv_Llm, x0 := 0, x1 := 27648, y1 := "dbtags_Sterowanie".SetupControlPompownia.r_Pv_Hlm, Ret_Val => "dbdane".act_Value_B6)
   END_RUNG
   // the same network as SCL:
   IF "AlwaysTRUE" THEN
       "dbdane".act_Value_B6 := "00_S_SclScaleLinearIntToReal"(x := "dbdane".PV_PER_B6,
                               yMin := 0.0,
                               yMax := 10.0,
                               y0 := "dbtags_Sterowanie".SetupControlPompownia.r_Pv_Llm,
                               x0 := 0,
                               x1 := 27648,
                               y1 := "dbtags_Sterowanie".SetupControlPompownia.r_Pv_Hlm);
   END_IF;
END_REGION

REGION Network 8: Ciśnienie magistrala strafa 1
   // Pomiar z czujnika B7  "Pompownia" - na wlocie do pompowni
   RUNG wire#powerrail
      Contact( "AlwaysTRUE" )
      "00_S_SclScaleLinearIntToReal"(x := "dbdane".PV_PER_B5, yMin := 0.0, yMax := 10.0, y0 := "dbtags_Sterowanie".SetupControlPompownia.r_Pv_Llm, x0 := 0, x1 := 27648, y1 := "dbtags_Sterowanie".SetupControlPompownia.r_Pv_Hlm, Ret_Val => "dbdane".act_Value_B5)
   END_RUNG
   // the same network as SCL:
   IF "AlwaysTRUE" THEN
       "dbdane".act_Value_B5 := "00_S_SclScaleLinearIntToReal"(x := "dbdane".PV_PER_B5,
                               yMin := 0.0,
                               yMax := 10.0,
                               y0 := "dbtags_Sterowanie".SetupControlPompownia.r_Pv_Llm,
                               x0 := 0,
                               x1 := 27648,
                               y1 := "dbtags_Sterowanie".SetupControlPompownia.r_Pv_Hlm);
   END_IF;
END_REGION

REGION Network 9: Poziom zbiornik nr 1
   // Pomiar poziomu w zbiorniku
   RUNG wire#powerrail
      Contact( "AlwaysTRUE" )
      "00_S_SclScaleLinearInt"(x := "dbdane".actSignalTank1, yMin := "dbtags_Sterowanie".Zbiorniki_sondy."Pv.LIm_Tank1", yMax := "dbtags_Sterowanie".Zbiorniki_sondy."Pv.HIm_Tank1", x0 := 0, y0 := "dbtags_Sterowanie".Zbiorniki_sondy."Pv.LIm_Tank1", x1 := 27648, y1 := "dbtags_Sterowanie".Zbiorniki_sondy."Pv.HIm_Tank1", Ret_Val => "dbdane".actValu_Tank1)
   END_RUNG
   // the same network as SCL:
   IF "AlwaysTRUE" THEN
       "dbdane".actValu_Tank1 := "00_S_SclScaleLinearInt"(x := "dbdane".actSignalTank1,
                               yMin := "dbtags_Sterowanie".Zbiorniki_sondy."Pv.LIm_Tank1",
                               yMax := "dbtags_Sterowanie".Zbiorniki_sondy."Pv.HIm_Tank1",
                               x0 := 0,
                               y0 := "dbtags_Sterowanie".Zbiorniki_sondy."Pv.LIm_Tank1",
                               x1 := 27648,
                               y1 := "dbtags_Sterowanie".Zbiorniki_sondy."Pv.HIm_Tank1");
   END_IF;
END_REGION

REGION Network 10: Poziom zbiornik nr 2
   // Pomiar poziomu w zbiorniku
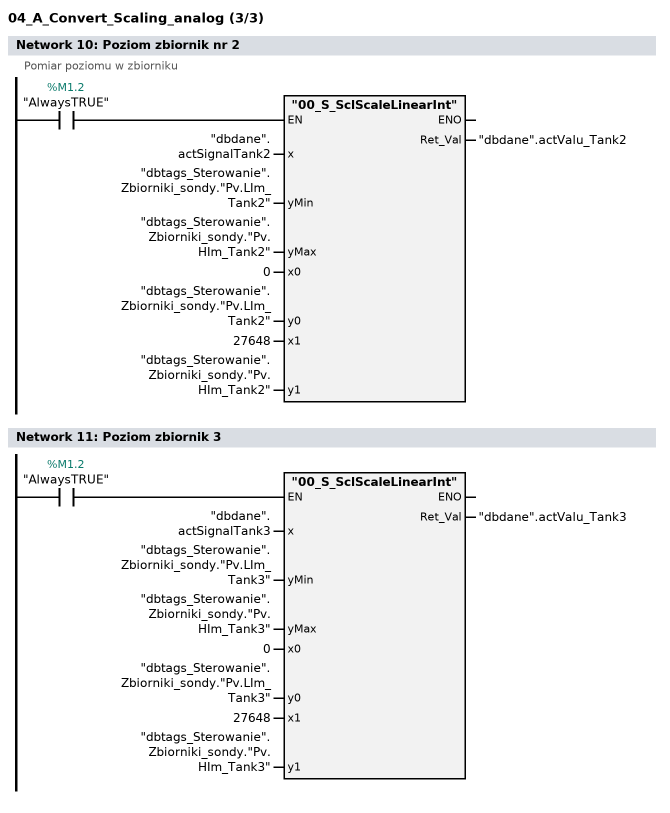
   RUNG wire#powerrail
      Contact( "AlwaysTRUE" )
      "00_S_SclScaleLinearInt"(x := "dbdane".actSignalTank2, yMin := "dbtags_Sterowanie".Zbiorniki_sondy."Pv.LIm_Tank2", yMax := "dbtags_Sterowanie".Zbiorniki_sondy."Pv.HIm_Tank2", x0 := 0, y0 := "dbtags_Sterowanie".Zbiorniki_sondy."Pv.LIm_Tank2", x1 := 27648, y1 := "dbtags_Sterowanie".Zbiorniki_sondy."Pv.HIm_Tank2", Ret_Val => "dbdane".actValu_Tank2)
   END_RUNG
   // the same network as SCL:
   IF "AlwaysTRUE" THEN
       "dbdane".actValu_Tank2 := "00_S_SclScaleLinearInt"(x := "dbdane".actSignalTank2,
                               yMin := "dbtags_Sterowanie".Zbiorniki_sondy."Pv.LIm_Tank2",
                               yMax := "dbtags_Sterowanie".Zbiorniki_sondy."Pv.HIm_Tank2",
                               x0 := 0,
                               y0 := "dbtags_Sterowanie".Zbiorniki_sondy."Pv.LIm_Tank2",
                               x1 := 27648,
                               y1 := "dbtags_Sterowanie".Zbiorniki_sondy."Pv.HIm_Tank2");
   END_IF;
END_REGION

REGION Network 11: Poziom zbiornik 3
   RUNG wire#powerrail
      Contact( "AlwaysTRUE" )
      "00_S_SclScaleLinearInt"(x := "dbdane".actSignalTank3, yMin := "dbtags_Sterowanie".Zbiorniki_sondy."Pv.LIm_Tank3", yMax := "dbtags_Sterowanie".Zbiorniki_sondy."Pv.HIm_Tank3", x0 := 0, y0 := "dbtags_Sterowanie".Zbiorniki_sondy."Pv.LIm_Tank3", x1 := 27648, y1 := "dbtags_Sterowanie".Zbiorniki_sondy."Pv.HIm_Tank3", Ret_Val => "dbdane".actValu_Tank3)
   END_RUNG
   // the same network as SCL:
   IF "AlwaysTRUE" THEN
       "dbdane".actValu_Tank3 := "00_S_SclScaleLinearInt"(x := "dbdane".actSignalTank3,
                               yMin := "dbtags_Sterowanie".Zbiorniki_sondy."Pv.LIm_Tank3",
                               yMax := "dbtags_Sterowanie".Zbiorniki_sondy."Pv.HIm_Tank3",
                               x0 := 0,
                               y0 := "dbtags_Sterowanie".Zbiorniki_sondy."Pv.LIm_Tank3",
                               x1 := 27648,
                               y1 := "dbtags_Sterowanie".Zbiorniki_sondy."Pv.HIm_Tank3");
   END_IF;
END_REGION
END_FUNCTION

FUNCTION "00_S_SclScaleLinearIntToReal" : Real
{ S7_Optimized_Access := 'TRUE' }
VERSION : 0.1
   VAR_INPUT 
      x : Int;
      yMin : Real;   // Granica minimalnej wartości fizycznej
      yMax : Real;   // Granica maxymalnej wartości fizycznej
      y0 : Real;   // Minimalna wartość wartości fizycznej (procesowej)
      x0 : Int;   // Minimalna wartość dla danego przetornika ADC zgodnie z dokumentacją Siemens
      x1 : Int;   // Maxymalna wartość dla danego przetornika ADC zgodnie z dokumentacją Siemens
      y1 : Real;   // Maxymalna wartość wartości fizycznej (procesowej)
   END_VAR

   VAR_TEMP 
      tempXreal : Real;
      tempX1real : Real;
      tempX0real : Real;
      tempYwert : Real;
   END_VAR


BEGIN
	#tempXreal := INT_TO_REAL(#x);
	#tempX0real := INT_TO_REAL(#x0);
	#tempX1real := INT_TO_REAL(#x1);
	
	IF (#x1 - #x0) = 0 OR (#x - #x0) = 0 OR (#y1 - #y0) = 0 OR #yMin > #yMax
	THEN
	    #tempYwert := 0;
	ELSE
	    #tempYwert := (#y1 - #y0) / (#tempX1real - #tempX0real) * (#tempXreal - #tempX0real) + #y0;
	END_IF;
	IF #tempYwert < #yMin THEN
	    #"00_S_SclScaleLinearIntToReal" := 0;
	ELSIF #tempYwert > #yMax THEN
	    #"00_S_SclScaleLinearIntToReal" := #yMax;
	ELSE
	    #"00_S_SclScaleLinearIntToReal" := #tempYwert;
	END_IF;
END_FUNCTION

FUNCTION "01_E_alarm handling" : Void   // FC10, LAD
TITLE = Boks Ready
{ S7_Optimized_Access := 'TRUE' }
AUTHOR : R.Tecmer
VERSION : 0.1
// Handling of alarms. Signaling and deleting
// stored: AutoNumber true, IsIECCheckEnabled false, SetENOAutomatically false, UDAEnableTagReadback false
   VAR_TEMP   // added for the SCL form of the ladder/FBD networks
      _w1 : Bool;
   END_VAR
BEGIN

REGION Network 1: Ready Inverters No1 No2
   // połączyłem bo usunięto drugi falownik
   // Jeśli brak gotowości to ustaw bity
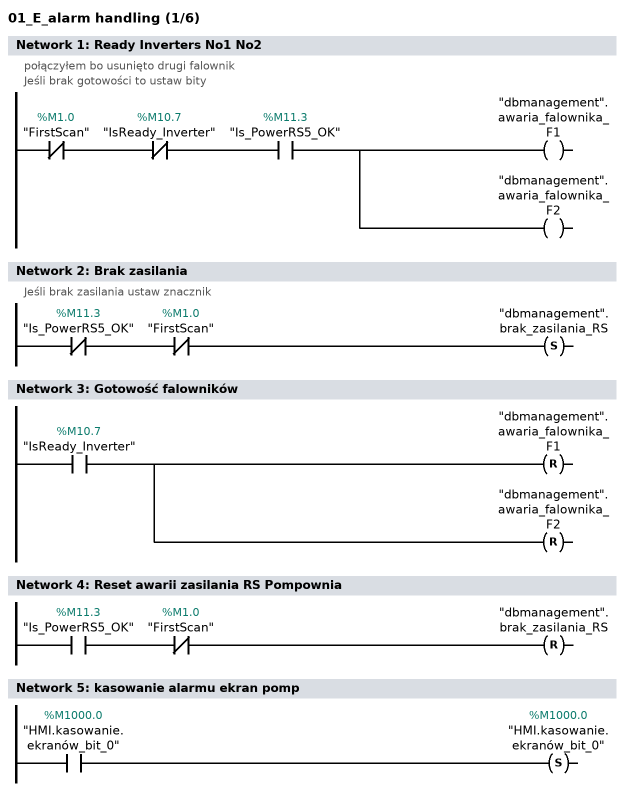
   RUNG wire#powerrail
      I_Contact( "FirstScan" )
      I_Contact( "IsReady_Inverter" )
      Contact( "Is_PowerRS5_OK" )
      wire#w1
      Coil( "dbmanagement".awaria_falownika_F1 )
   END_RUNG
   RUNG wire#w1
      Coil( "dbmanagement".awaria_falownika_F2 )
   END_RUNG
   // the same network as SCL:
   "dbmanagement".awaria_falownika_F1 := NOT "FirstScan" AND NOT "IsReady_Inverter" AND "Is_PowerRS5_OK";
   "dbmanagement".awaria_falownika_F2 := "dbmanagement".awaria_falownika_F1;
END_REGION

REGION Network 2: Brak zasilania
   // Jeśli brak zasilania ustaw znacznik
   RUNG wire#powerrail
      I_Contact( "Is_PowerRS5_OK" )
      I_Contact( "FirstScan" )
      S_Coil( "dbmanagement".brak_zasilania_RS )
   END_RUNG
   // the same network as SCL:
   IF NOT "Is_PowerRS5_OK" AND NOT "FirstScan" THEN "dbmanagement".brak_zasilania_RS := TRUE; END_IF;
END_REGION

REGION Network 3: Gotowość falowników
   RUNG wire#powerrail
      Contact( "IsReady_Inverter" )
      wire#w1
      R_Coil( "dbmanagement".awaria_falownika_F1 )
   END_RUNG
   RUNG wire#w1
      R_Coil( "dbmanagement".awaria_falownika_F2 )
   END_RUNG
   // the same network as SCL:
   IF "IsReady_Inverter" THEN
       "dbmanagement".awaria_falownika_F1 := FALSE;
       "dbmanagement".awaria_falownika_F2 := FALSE;
   END_IF;
END_REGION

REGION Network 4: Reset awarii zasilania RS Pompownia
   RUNG wire#powerrail
      Contact( "Is_PowerRS5_OK" )
      I_Contact( "FirstScan" )
      R_Coil( "dbmanagement".brak_zasilania_RS )
   END_RUNG
   // the same network as SCL:
   IF "Is_PowerRS5_OK" AND NOT "FirstScan" THEN "dbmanagement".brak_zasilania_RS := FALSE; END_IF;
END_REGION

REGION Network 5: kasowanie alarmu ekran pomp
   RUNG wire#powerrail
      Contact( "HMI.kasowanie.ekranów_bit_0" )
      S_Coil( "HMI.kasowanie.ekranów_bit_0" )
   END_RUNG
   // the same network as SCL:
   IF "HMI.kasowanie.ekranów_bit_0" THEN "HMI.kasowanie.ekranów_bit_0" := TRUE; END_IF;
END_REGION

REGION Network 6: Procedura kasowania alarmu - interakcja z SCADA P1 P2 P3 P4
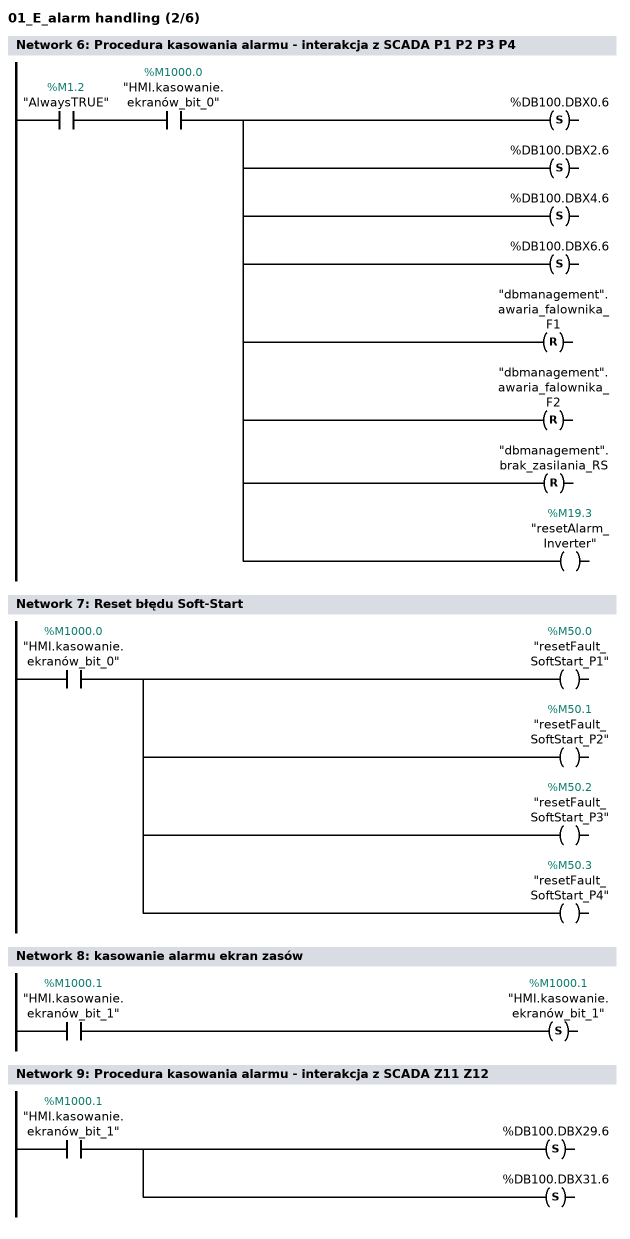
   RUNG wire#powerrail
      Contact( "AlwaysTRUE" )
      Contact( "HMI.kasowanie.ekranów_bit_0" )
      wire#w1
      S_Coil( %DB100.DBX0.6 )
   END_RUNG
   RUNG wire#w1
      S_Coil( %DB100.DBX2.6 )
   END_RUNG
   RUNG wire#w1
      S_Coil( %DB100.DBX4.6 )
   END_RUNG
   RUNG wire#w1
      S_Coil( %DB100.DBX6.6 )
   END_RUNG
   RUNG wire#w1
      R_Coil( "dbmanagement".awaria_falownika_F1 )
   END_RUNG
   RUNG wire#w1
      R_Coil( "dbmanagement".awaria_falownika_F2 )
   END_RUNG
   RUNG wire#w1
      R_Coil( "dbmanagement".brak_zasilania_RS )
   END_RUNG
   RUNG wire#w1
      Coil( "resetAlarm_Inverter" )
   END_RUNG
   // the same network as SCL:
   #_w1 := "AlwaysTRUE" AND "HMI.kasowanie.ekranów_bit_0";
   IF #_w1 THEN
       %DB100.DBX0.6 := TRUE;
       %DB100.DBX2.6 := TRUE;
       %DB100.DBX4.6 := TRUE;
       %DB100.DBX6.6 := TRUE;
       "dbmanagement".awaria_falownika_F1 := FALSE;
       "dbmanagement".awaria_falownika_F2 := FALSE;
       "dbmanagement".brak_zasilania_RS := FALSE;
   END_IF;
   "resetAlarm_Inverter" := #_w1;
END_REGION

REGION Network 7: Reset błędu Soft-Start
   RUNG wire#powerrail
      Contact( "HMI.kasowanie.ekranów_bit_0" )
      wire#w1
      Coil( "resetFault_SoftStart_P1" )
   END_RUNG
   RUNG wire#w1
      Coil( "resetFault_SoftStart_P2" )
   END_RUNG
   RUNG wire#w1
      Coil( "resetFault_SoftStart_P3" )
   END_RUNG
   RUNG wire#w1
      Coil( "resetFault_SoftStart_P4" )
   END_RUNG
   // the same network as SCL:
   "resetFault_SoftStart_P1" := "HMI.kasowanie.ekranów_bit_0";
   "resetFault_SoftStart_P2" := "HMI.kasowanie.ekranów_bit_0";
   "resetFault_SoftStart_P3" := "HMI.kasowanie.ekranów_bit_0";
   "resetFault_SoftStart_P4" := "HMI.kasowanie.ekranów_bit_0";
END_REGION

REGION Network 8: kasowanie alarmu ekran zasów
   RUNG wire#powerrail
      Contact( "HMI.kasowanie.ekranów_bit_1" )
      S_Coil( "HMI.kasowanie.ekranów_bit_1" )
   END_RUNG
   // the same network as SCL:
   IF "HMI.kasowanie.ekranów_bit_1" THEN "HMI.kasowanie.ekranów_bit_1" := TRUE; END_IF;
END_REGION

REGION Network 9: Procedura kasowania alarmu - interakcja z SCADA Z11 Z12
   RUNG wire#powerrail
      Contact( "HMI.kasowanie.ekranów_bit_1" )
      wire#w1
      S_Coil( %DB100.DBX29.6 )
   END_RUNG
   RUNG wire#w1
      S_Coil( %DB100.DBX31.6 )
   END_RUNG
   // the same network as SCL:
   IF "HMI.kasowanie.ekranów_bit_1" THEN
       %DB100.DBX29.6 := TRUE;
       %DB100.DBX31.6 := TRUE;
   END_IF;
END_REGION

REGION Network 10: Alarm Fault Modbus RTU
   // Alarm błędu komunikacji modbus
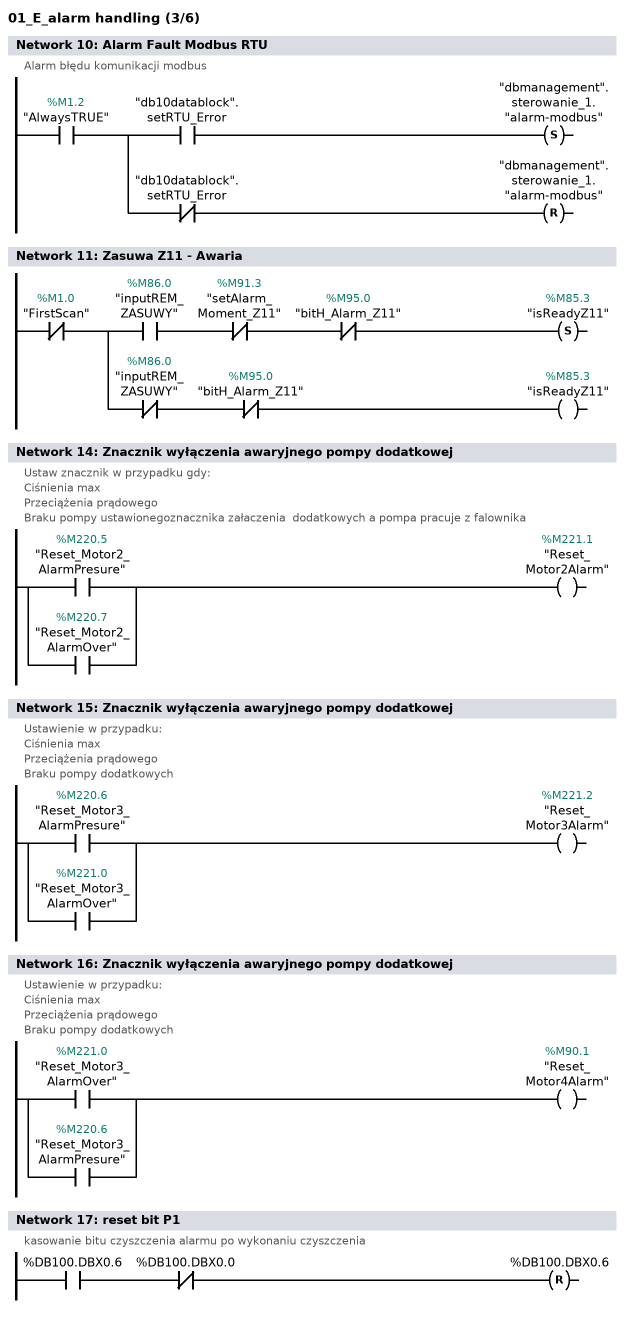
   RUNG wire#powerrail
      Contact( "AlwaysTRUE" )
      wire#w1
      Contact( "db10datablock".setRTU_Error )
      S_Coil( "dbmanagement".sterowanie_1."alarm-modbus" )
   END_RUNG
   RUNG wire#w1
      I_Contact( "db10datablock".setRTU_Error )
      R_Coil( "dbmanagement".sterowanie_1."alarm-modbus" )
   END_RUNG
   // the same network as SCL:
   IF "AlwaysTRUE" AND "db10datablock".setRTU_Error THEN
       "dbmanagement".sterowanie_1."alarm-modbus" := TRUE;
   END_IF;
   IF "AlwaysTRUE" AND NOT "db10datablock".setRTU_Error THEN
       "dbmanagement".sterowanie_1."alarm-modbus" := FALSE;
   END_IF;
END_REGION

REGION Network 11: Zasuwa Z11 - Awaria
   RUNG wire#powerrail
      I_Contact( "FirstScan" )
      wire#w1
      Contact( "inputREM_ZASUWY" )
      I_Contact( "setAlarm_Moment_Z11" )
      I_Contact( "bitH_Alarm_Z11" )
      S_Coil( "isReadyZ11" )
   END_RUNG
   RUNG wire#w1
      I_Contact( "inputREM_ZASUWY" )
      I_Contact( "bitH_Alarm_Z11" )
      Coil( "isReadyZ11" )
   END_RUNG
   // the same network as SCL:
   IF NOT "FirstScan" AND "inputREM_ZASUWY" AND NOT "setAlarm_Moment_Z11" AND NOT "bitH_Alarm_Z11" THEN
       "isReadyZ11" := TRUE;
   END_IF;
   "isReadyZ11" := NOT "FirstScan" AND NOT "inputREM_ZASUWY" AND NOT "bitH_Alarm_Z11";
END_REGION

REGION Network 12 (SCL): Z11 znacznik alarmu od momentówki w trybie zdalnym (aut/mamnual)
   IF  "inputAwariaMomentZ11" = False THEN
     // Ustaw alarm od momentu
     "setAlarm_Moment_Z11" := TRUE;
   ELSE
     "setAlarm_Moment_Z11" := FALSE;
     ;
   END_IF;
END_REGION

REGION Network 13 (SCL): Ustaw brak gotowości Z11
   IF "setAlarm_Moment_Z11" = TRUE OR "bitH_Alarm_Z11" THEN
     // Ustaw Alarm
     "isReadyZ11" := FALSE;

     ;
   END_IF;
END_REGION

REGION Network 14: Znacznik wyłączenia awaryjnego pompy dodatkowej
   // Ustaw znacznik w przypadku gdy:
   // Ciśnienia max
   // Przeciążenia prądowego
   // Braku pompy ustawionegoznacznika załaczenia  dodatkowych a pompa pracuje z falownika
   RUNG wire#powerrail
      Contact( "Reset_Motor2_AlarmPresure" )
      wire#w1
      Coil( "Reset_Motor2Alarm" )
   END_RUNG
   RUNG wire#powerrail
      Contact( "Reset_Motor2_AlarmOver" )
   END_RUNG wire#w1
   // the same network as SCL:
   "Reset_Motor2Alarm" := "Reset_Motor2_AlarmPresure" OR "Reset_Motor2_AlarmOver";
END_REGION

REGION Network 15: Znacznik wyłączenia awaryjnego pompy dodatkowej
   // Ustawienie w przypadku:
   // Ciśnienia max
   // Przeciążenia prądowego
   // Braku pompy dodatkowych
   RUNG wire#powerrail
      Contact( "Reset_Motor3_AlarmPresure" )
      wire#w1
      Coil( "Reset_Motor3Alarm" )
   END_RUNG
   RUNG wire#powerrail
      Contact( "Reset_Motor3_AlarmOver" )
   END_RUNG wire#w1
   // the same network as SCL:
   "Reset_Motor3Alarm" := "Reset_Motor3_AlarmPresure" OR "Reset_Motor3_AlarmOver";
END_REGION

REGION Network 16: Znacznik wyłączenia awaryjnego pompy dodatkowej
   // Ustawienie w przypadku:
   // Ciśnienia max
   // Przeciążenia prądowego
   // Braku pompy dodatkowych
   RUNG wire#powerrail
      Contact( "Reset_Motor3_AlarmOver" )
      wire#w1
      Coil( "Reset_Motor4Alarm" )
   END_RUNG
   RUNG wire#powerrail
      Contact( "Reset_Motor3_AlarmPresure" )
   END_RUNG wire#w1
   // the same network as SCL:
   "Reset_Motor4Alarm" := "Reset_Motor3_AlarmOver" OR "Reset_Motor3_AlarmPresure";
END_REGION

REGION Network 17: reset bit P1
   // kasowanie bitu czyszczenia alarmu po wykonaniu czyszczenia
   RUNG wire#powerrail
      Contact( %DB100.DBX0.6 )
      I_Contact( %DB100.DBX0.0 )
      R_Coil( %DB100.DBX0.6 )
   END_RUNG
   // the same network as SCL:
   IF %DB100.DBX0.6 AND NOT %DB100.DBX0.0 THEN %DB100.DBX0.6 := FALSE; END_IF;
END_REGION

REGION Network 18: reset bit P2
   // kasowanie bitu czyszczenia alarmu po wykonaniu czyszczenia
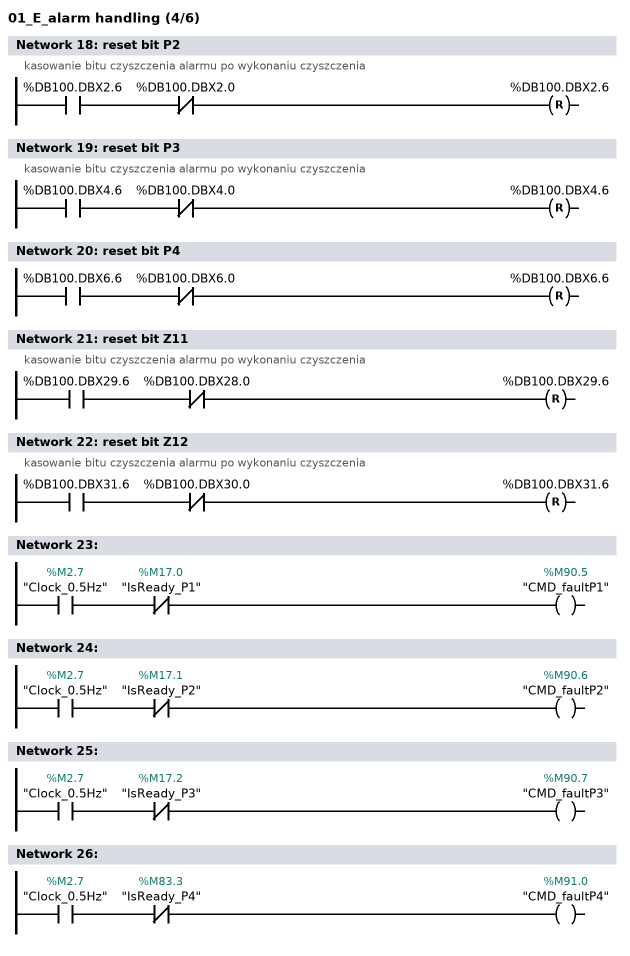
   RUNG wire#powerrail
      Contact( %DB100.DBX2.6 )
      I_Contact( %DB100.DBX2.0 )
      R_Coil( %DB100.DBX2.6 )
   END_RUNG
   // the same network as SCL:
   IF %DB100.DBX2.6 AND NOT %DB100.DBX2.0 THEN %DB100.DBX2.6 := FALSE; END_IF;
END_REGION

REGION Network 19: reset bit P3
   // kasowanie bitu czyszczenia alarmu po wykonaniu czyszczenia
   RUNG wire#powerrail
      Contact( %DB100.DBX4.6 )
      I_Contact( %DB100.DBX4.0 )
      R_Coil( %DB100.DBX4.6 )
   END_RUNG
   // the same network as SCL:
   IF %DB100.DBX4.6 AND NOT %DB100.DBX4.0 THEN %DB100.DBX4.6 := FALSE; END_IF;
END_REGION

REGION Network 20: reset bit P4
   RUNG wire#powerrail
      Contact( %DB100.DBX6.6 )
      I_Contact( %DB100.DBX6.0 )
      R_Coil( %DB100.DBX6.6 )
   END_RUNG
   // the same network as SCL:
   IF %DB100.DBX6.6 AND NOT %DB100.DBX6.0 THEN %DB100.DBX6.6 := FALSE; END_IF;
END_REGION

REGION Network 21: reset bit Z11
   // kasowanie bitu czyszczenia alarmu po wykonaniu czyszczenia
   RUNG wire#powerrail
      Contact( %DB100.DBX29.6 )
      I_Contact( %DB100.DBX28.0 )
      R_Coil( %DB100.DBX29.6 )
   END_RUNG
   // the same network as SCL:
   IF %DB100.DBX29.6 AND NOT %DB100.DBX28.0 THEN %DB100.DBX29.6 := FALSE; END_IF;
END_REGION

REGION Network 22: reset bit Z12
   // kasowanie bitu czyszczenia alarmu po wykonaniu czyszczenia
   RUNG wire#powerrail
      Contact( %DB100.DBX31.6 )
      I_Contact( %DB100.DBX30.0 )
      R_Coil( %DB100.DBX31.6 )
   END_RUNG
   // the same network as SCL:
   IF %DB100.DBX31.6 AND NOT %DB100.DBX30.0 THEN %DB100.DBX31.6 := FALSE; END_IF;
END_REGION

REGION Network 23
   RUNG wire#powerrail
      Contact( "Clock_0.5Hz" )
      I_Contact( "IsReady_P1" )
      Coil( "CMD_faultP1" )
   END_RUNG
   // the same network as SCL:
   "CMD_faultP1" := "Clock_0.5Hz" AND NOT "IsReady_P1";
END_REGION

REGION Network 24
   RUNG wire#powerrail
      Contact( "Clock_0.5Hz" )
      I_Contact( "IsReady_P2" )
      Coil( "CMD_faultP2" )
   END_RUNG
   // the same network as SCL:
   "CMD_faultP2" := "Clock_0.5Hz" AND NOT "IsReady_P2";
END_REGION

REGION Network 25
   RUNG wire#powerrail
      Contact( "Clock_0.5Hz" )
      I_Contact( "IsReady_P3" )
      Coil( "CMD_faultP3" )
   END_RUNG
   // the same network as SCL:
   "CMD_faultP3" := "Clock_0.5Hz" AND NOT "IsReady_P3";
END_REGION

REGION Network 26
   RUNG wire#powerrail
      Contact( "Clock_0.5Hz" )
      I_Contact( "IsReady_P4" )
      Coil( "CMD_faultP4" )
   END_RUNG
   // the same network as SCL:
   "CMD_faultP4" := "Clock_0.5Hz" AND NOT "IsReady_P4";
END_REGION

REGION Network 27: Przełączanie pomiary Hz Modba / Analog
   // Jesli awaria Modbus RTU aktualna wartość Hz pobierana bedzie z wejścia analogowego falownia (wyjście AQ PLC)
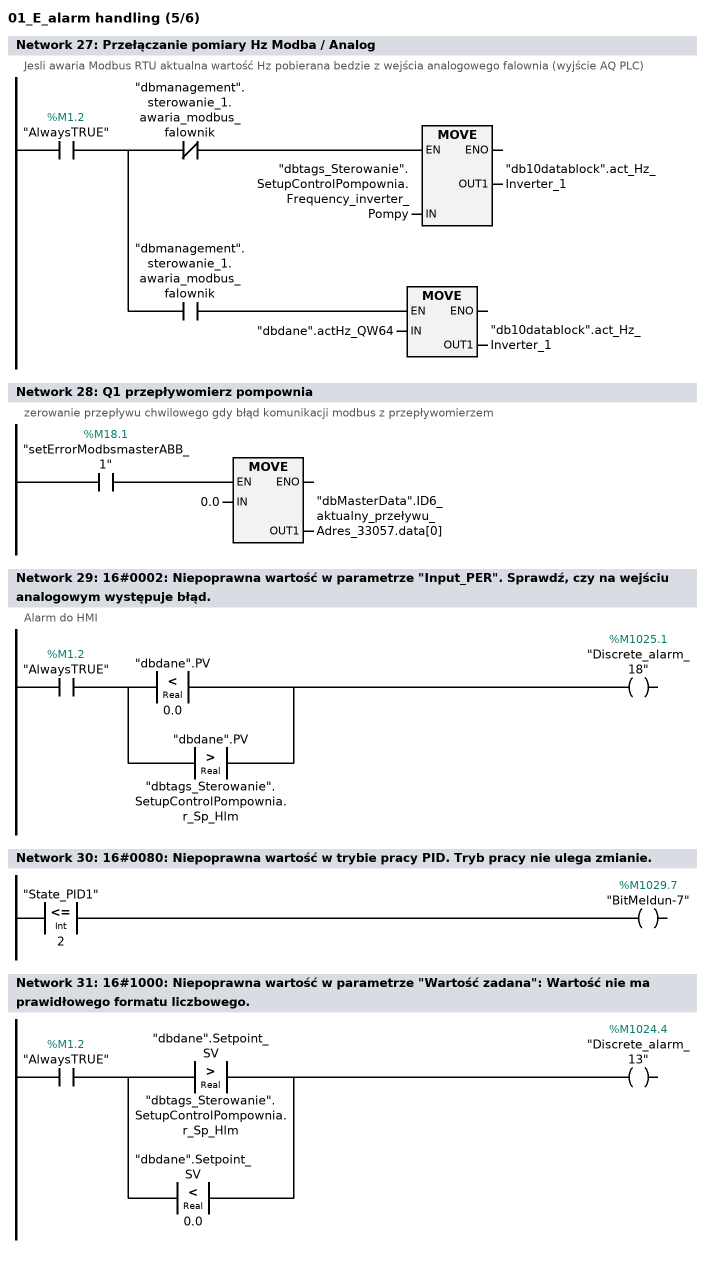
   RUNG wire#powerrail
      Contact( "AlwaysTRUE" )
      wire#w1
      I_Contact( "dbmanagement".sterowanie_1.awaria_modbus_falownik )
      Move(in := "dbtags_Sterowanie".SetupControlPompownia.Frequency_inverter_Pompy, out1 => "db10datablock".act_Hz_Inverter_1)
   END_RUNG
   RUNG wire#w1
      Contact( "dbmanagement".sterowanie_1.awaria_modbus_falownik )
      Move(in := "dbdane".actHz_QW64, out1 => "db10datablock".act_Hz_Inverter_1)
   END_RUNG
   // the same network as SCL:
   IF "AlwaysTRUE" AND NOT "dbmanagement".sterowanie_1.awaria_modbus_falownik THEN
       "db10datablock".act_Hz_Inverter_1 := "dbtags_Sterowanie".SetupControlPompownia.Frequency_inverter_Pompy;
   END_IF;
   IF "AlwaysTRUE" AND "dbmanagement".sterowanie_1.awaria_modbus_falownik THEN
       "db10datablock".act_Hz_Inverter_1 := "dbdane".actHz_QW64;
   END_IF;
END_REGION

REGION Network 28: Q1 przepływomierz pompownia
   // zerowanie przepływu chwilowego gdy błąd komunikacji modbus z przepływomierzem
   RUNG wire#powerrail
      Contact( "setErrorModbsmasterABB_1" )
      { S7_GenerateENO := "TRUE" } Move(in := 0.0, out1 => "dbMasterData".ID6_aktualny_przeływu_Adres_33057.data[0])
   END_RUNG
   // the same network as SCL:
   IF "setErrorModbsmasterABB_1" THEN
       "dbMasterData".ID6_aktualny_przeływu_Adres_33057.data[0] := 0.0;
   END_IF;
END_REGION

REGION Network 29: 16#0002: Niepoprawna wartość w parametrze "Input_PER". Sprawdź, czy na wejściu analogowym występuje błąd.
   // Alarm do HMI
   RUNG wire#powerrail
      Contact( "AlwaysTRUE" )
      wire#w1
      { S7_Templates := "SrcType := Real" } LT_Contact(in1 := "dbdane".PV, in2 := 0.0)
      wire#w2
      Coil( "Discrete_alarm_18" )
   END_RUNG
   RUNG wire#w1
      { S7_Templates := "SrcType := Real" } GT_Contact(in1 := "dbdane".PV, in2 := "dbtags_Sterowanie".SetupControlPompownia.r_Sp_Hlm)
   END_RUNG wire#w2
   // the same network as SCL:
   "Discrete_alarm_18" := "AlwaysTRUE" AND (("dbdane".PV < 0.0) OR ("dbdane".PV > "dbtags_Sterowanie".SetupControlPompownia.r_Sp_Hlm));
END_REGION

REGION Network 30: 16#0080: Niepoprawna wartość w trybie pracy PID. Tryb pracy nie ulega zmianie.
   RUNG wire#powerrail
      { S7_Templates := "SrcType := Int" } LE_Contact(in1 := "State_PID1", in2 := 2)
      Coil( "BitMeldun-7" )
   END_RUNG
   // the same network as SCL:
   "BitMeldun-7" := "State_PID1" <= 2;
END_REGION

REGION Network 31: 16#1000: Niepoprawna wartość w parametrze "Wartość zadana": Wartość nie ma prawidłowego formatu liczbowego.
   RUNG wire#powerrail
      Contact( "AlwaysTRUE" )
      wire#w1
      { S7_Templates := "SrcType := Real" } GT_Contact(in1 := "dbdane".Setpoint_SV, in2 := "dbtags_Sterowanie".SetupControlPompownia.r_Sp_Hlm)
      wire#w2
      Coil( "Discrete_alarm_13" )
   END_RUNG
   RUNG wire#w1
      { S7_Templates := "SrcType := Real" } LT_Contact(in1 := "dbdane".Setpoint_SV, in2 := 0.0)
   END_RUNG wire#w2
   // the same network as SCL:
   "Discrete_alarm_13" := "AlwaysTRUE" AND (("dbdane".Setpoint_SV > "dbtags_Sterowanie".SetupControlPompownia.r_Sp_Hlm) OR ("dbdane".Setpoint_SV < 0.0));
END_REGION

REGION Network 32: alarm magistrala niskie ciśnienie
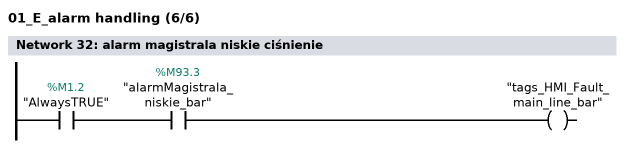
   RUNG wire#powerrail
      Contact( "AlwaysTRUE" )
      Contact( "alarmMagistrala_niskie_bar" )
      Coil( "tags_HMI_Fault_main_line_bar" )
   END_RUNG
   // the same network as SCL:
   "tags_HMI_Fault_main_line_bar" := "AlwaysTRUE" AND "alarmMagistrala_niskie_bar";
END_REGION
END_FUNCTION

FUNCTION_BLOCK "01_E_bar max"
TITLE = Control press oxygen 
{ S7_Optimized_Access := 'TRUE' }
AUTHOR : rtecmer
VERSION : 0.1
//Kontrola ciśnienia w rurociągu. Sterowanie ograniczeniem wydajności falownika w przypadku przekroczenia ciśnienia max
   VAR_INPUT 
      dane_Pressure_bar : Real;   // Aktualne ciśnienie w rurociągu
      Press_Max { ExternalAccessible := 'False'; ExternalVisible := 'False'; ExternalWritable := 'False'} : Real;   // Ciśnienie graniczne max
   END_VAR

   VAR_OUTPUT 
      bar_max : Bool;   // Bit sygnału alarm ciśnienie za wysokie w rurociągu
   END_VAR

   VAR_TEMP 
      Temp_Press_max : Bool;   // Znacznik pomocniczy
   END_VAR


BEGIN
	(*
	//=============================================================================
	//(JZWiK S.A Radosław Tecmer)
	//(c)Copyright (2022) All Rights Reserved
	//-----------------------------------------------------------------------------
	//Testowane z:   (system docelowy z  FW 4.4)
	//Pakiet inżynierski:   TIA Portal (V16 Update 5)
	//Ograniczenia:  ( - )
	//Wymagania:  (minimalne S7-1200 CPU 1215C FW 4.2 .)
	//Funkcjonalnośc: (Kontrola cisnienia tłoczenia z wystawieniem 
	                   sygnału przekroczenia cisnieie max)
	//-----------------------------------------------------------------------------
	//Zmainy wprowadzone:
	//Wersja  Data       Osoba wprowadzająca zmiany - ekspert
	//01.00.00 09.03.2022 (Tecmer Radosław - twórca) Pieresza wersja 01.00.00
	//=============================================================================
	*)
	
	REGION Control Press
	  // Porównanie aktualnego z Max
	  IF #dane_Pressure_bar > #Press_Max THEN
	    // Ustawienie znacznika jeśli Act > Max
	    #Temp_Press_max := TRUE;
	  ELSE
	    #Temp_Press_max := FALSE;
	    ;
	  END_IF;
	  
	 "IEC_Timer_PressO2_Max_DB".TON(IN:= #Temp_Press_max,
	                                 PT:= T#15S,
	                                 Q=> #bar_max);
	  
	  
	END_REGION
	
END_FUNCTION_BLOCK

FUNCTION "01_E_stop_additional_pump_max_bar" : Void   // FC13, LAD
TITLE = Stopping pumps due to bar max
{ S7_Optimized_Access := 'TRUE' }
AUTHOR : rtecmer
VERSION : 0.1
// Funkcja awaryjnego zatrzymania pomop z powodu ciśnienie max w przewodzie tłocznym
// stored: AutoNumber true, IsIECCheckEnabled false, SetENOAutomatically false, UDAEnableTagReadback false
   VAR_INPUT
      is_bar_max : Bool;   // znacznik alarmu ciśnienia max w tłocznym
      is_network_run_P1 : Bool;   // potwierdzenie pracy pompy z sieci
      is_network_run_P2 : Bool;   // potwierdzenie pracy pompy z sieci
      is_network_run_P3 : Bool;   // potwierdzenie pracy pompy z sieci
   END_VAR
   VAR_IN_OUT
      setCMD_P1 : Bool;   // znacznik sterowania pompą z sieci
      setCMD_P2 : Bool;   // znacznik sterowania pompą z sieci
      setCMD_P3 : Bool;   // znacznik sterowania pompą z sieci
   END_VAR
BEGIN

REGION Network 1: znacznik sterowania pompą z sieci
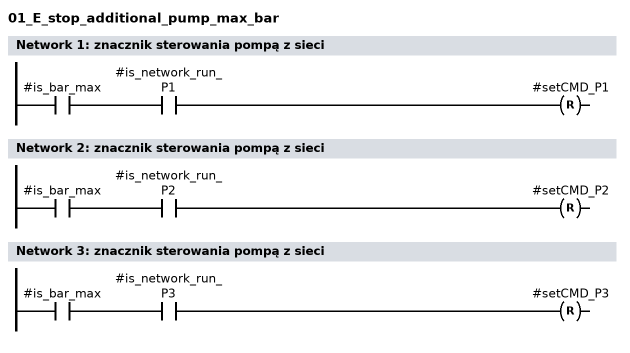
   RUNG wire#powerrail
      Contact( #is_bar_max )
      Contact( #is_network_run_P1 )
      R_Coil( #setCMD_P1 )
   END_RUNG
   // the same network as SCL:
   IF #is_bar_max AND #is_network_run_P1 THEN #setCMD_P1 := FALSE; END_IF;
END_REGION

REGION Network 2: znacznik sterowania pompą z sieci
   RUNG wire#powerrail
      Contact( #is_bar_max )
      Contact( #is_network_run_P2 )
      R_Coil( #setCMD_P2 )
   END_RUNG
   // the same network as SCL:
   IF #is_bar_max AND #is_network_run_P2 THEN #setCMD_P2 := FALSE; END_IF;
END_REGION

REGION Network 3: znacznik sterowania pompą z sieci
   RUNG wire#powerrail
      Contact( #is_bar_max )
      Contact( #is_network_run_P3 )
      R_Coil( #setCMD_P3 )
   END_RUNG
   // the same network as SCL:
   IF #is_bar_max AND #is_network_run_P3 THEN #setCMD_P3 := FALSE; END_IF;
END_REGION
END_FUNCTION

FUNCTION_BLOCK "06_M_Control Hz safe mode from bar Max"
TITLE = Handing Oxygen Pressure Max
{ S7_Optimized_Access := 'TRUE' }
AUTHOR : rtecmer
VERSION : 0.1
//Sterowanie wydajnością invertera KDN w czasie wystąpienia alarmu od ciśnienia, przeciążenia
   VAR_INPUT 
      Value_Max : Bool;   // Znacznik Alarmowej wartości
      My_1Hz : Bool;
      Act_Hz : Real;   // Aktualne Hz przechwycone
      IsMotor2Set : Bool;   // Znacznik pierwszej pompy dodatkowej
      IsMotor3Set : Bool;   // Znacznik drugiej pompy dodatkowej
      IsMotor4Set : Bool;   // Znacznik trzeciej pompy dodatkowej
      IsReadyinverter1 : Bool;   // Gotowość falownika 1
   END_VAR

   VAR_OUTPUT 
      Value_Manual_Hz : Real := 10.0;   // Wartość procentowa [%}  Hz zadawanych w trybie awaryjnym
      Rst_Motor2 : Bool;   // Znacznik wyłaczenia awayjnego dodatkowej pompy pierwszej
      Rst_Motor3 : Bool;   // Znacznik wyłaczenia awayjnego dodatkowej pompy drugiej
      Rst_Motor4 : Bool;   // Znacznik wyłaczenia awayjnego dodatkowej pompy drugiej
      Rst_Driver : Bool := false;   // Znacznik wyłaczenia awayjnego
   END_VAR

   VAR 
      set_NewValue { ExternalAccessible := 'False'; ExternalVisible := 'False'; ExternalWritable := 'False'} : Bool;
      index { ExternalAccessible := 'False'; ExternalVisible := 'False'; ExternalWritable := 'False'} : Bool;
      CV { ExternalAccessible := 'False'; ExternalVisible := 'False'; ExternalWritable := 'False'} : Int;
      load_cunt { ExternalAccessible := 'False'; ExternalVisible := 'False'; ExternalWritable := 'False'} : Bool;
      tmp_Hz { ExternalAccessible := 'False'; ExternalVisible := 'False'; ExternalWritable := 'False'} : Real;   // Wartość Hz zatrzaśnięta do obliczeń
      cnt_Hz { ExternalAccessible := 'False'; ExternalVisible := 'False'; ExternalWritable := 'False'} : Real;   // Zmienna Hz do przeliczania w procesie sterowani podczas awarii
      mem_Triger_Alarm { ExternalAccessible := 'False'; ExternalVisible := 'False'; ExternalWritable := 'False'} : Bool;   // Pamięć zbocza narastającego wytąpienia alarmu
   END_VAR

   VAR CONSTANT 
      PV : Int := 5;   // Wartość procentowa licznika ładowanego dla Generacji wartości [%] Hz
   END_VAR


BEGIN
	(*
	Kontrola wartości zadanej Hz w trybie pracy awaryjnej od max 
	ciśnienia  w przewodzie
	*)
	
